LIN {X 0,Y 607.23,Z 1025.741,A -85,B 0,C 180,E1 27746.767,E2 27746.767} C_VEL
LIN {X 0,Y 605.649,Z 1047.101,A -85,B 0,C 180,E1 27745.787,E2 27745.787} C_VEL
LIN {X 0,Y 604.017,Z 1067.74,A -85,B 0,C 180,E1 27744.656,E2 27744.656} C_VEL
LIN {X 0,Y 602.404,Z 1085.974,A -85,B 0,C 180,E1 27743.476,E2 27743.476} C_VEL
LIN {X 0,Y 600.536,Z 1105.985,A -85,B 0,C 180,E1 27741.965,E2 27741.965} C_VEL
LIN {X 0,Y 598.945,Z 1123.019,A -85,B 0,C 180,E1 27740.472,E2 27740.472} C_VEL
LIN {X 0,Y 597.317,Z 1139.909,A -85,B 0,C 180,E1 27738.748,E2 27738.748} C_VEL
LIN {X 0,Y 595.864,Z 1155.688,A -85,B 0,C 180,E1 27736.876,E2 27736.876} C_VEL
LIN {X 0,Y 594.758,Z 1168.565,A -85,B 0,C 180,E1 27735.105,E2 27735.105} C_VEL
LIN {X 0,Y 593.832,Z 1180.293,A -85,B 0,C 180,E1 27733.238,E2 27733.238} C_VEL
LIN {X 0,Y 593.073,Z 1191.366,A -85,B 0,C 180,E1 27731.18,E2 27731.18} C_VEL
LIN {X 0,Y 592.512,Z 1201.281,A -85,B 0,C 180,E1 27728.932,E2 27728.932} C_VEL
LIN {X 0,Y 592.226,Z 1208.03,A -85,B 0,C 180,E1 27727.08,E2 27727.08} C_VEL
LIN {X 0,Y 592.061,Z 1213.419,A -85,B 0,C 180,E1 27725.33,E2 27725.33} C_VEL
LIN {X 0,Y 591.966,Z 1217.736,A -85,B 0,C 180,E1 27723.583,E2 27723.583} C_VEL
LIN {X 0,Y 591.922,Z 1221.023,A -85,B 0,C 180,E1 27721.839,E2 27721.839} C_VEL
LIN {X 0,Y 591.917,Z 1223.391,A -85,B 0,C 180,E1 27720,E2 27720} C_VEL
LIN {X 0,Y 591.915,Z 1224.654,A -85,B 0,C 180,E1 27718.161,E2 27718.161} C_VEL
LIN {X 0,Y 591.912,Z 1224.844,A -85,B 0,C 180,E1 27716.417,E2 27716.417} C_VEL
LIN {X 0,Y 591.911,Z 1224.051,A -85,B 0,C 180,E1 27714.669,E2 27714.669} C_VEL
LIN {X 0,Y 591.924,Z 1222.118,A -85,B 0,C 180,E1 27712.819,E2 27712.819} C_VEL
LIN {X 0,Y 591.947,Z 1219.241,A -85,B 0,C 180,E1 27711.06,E2 27711.06} C_VEL
LIN {X 0,Y 592.007,Z 1215.307,A -85,B 0,C 180,E1 27709.293,E2 27709.293} C_VEL
LIN {X 0,Y 592.15,Z 1210.275,A -85,B 0,C 180,E1 27707.518,E2 27707.518} C_VEL
LIN {X 0,Y 592.391,Z 1203.803,A -85,B 0,C 180,E1 27705.634,E2 27705.634} C_VEL
LIN {X 0,Y 592.739,Z 1196.926,A -85,B 0,C 180,E1 27703.939,E2 27703.939} C_VEL
LIN {X 0,Y 593.244,Z 1188.823,A -85,B 0,C 180,E1 27702.231,E2 27702.231} C_VEL
LIN {X 0,Y 594.061,Z 1177.572,A -85,B 0,C 180,E1 27700.201,E2 27700.201} C_VEL
LIN {X 0,Y 595.167,Z 1163.645,A -85,B 0,C 180,E1 27698.101,E2 27698.101} C_VEL
LIN {X 0,Y 596.308,Z 1150.164,A -85,B 0,C 180,E1 27696.374,E2 27696.374} C_VEL
LIN {X 0,Y 597.658,Z 1135.085,A -85,B 0,C 180,E1 27694.694,E2 27694.694} C_VEL
LIN {X 0,Y 599.006,Z 1119.589,A -85,B 0,C 180,E1 27693.211,E2 27693.211} C_VEL
LIN {X 0,Y 600.574,Z 1100.912,A -85,B 0,C 180,E1 27691.673,E2 27691.673} C_VEL
LIN {X 0,Y 602.005,Z 1082.997,A -85,B 0,C 180,E1 27690.411,E2 27690.411} C_VEL
LIN {X 0,Y 603.301,Z 1064.426,A -85,B 0,C 180,E1 27689.305,E2 27689.305} C_VEL
LIN {X 0,Y 604.533,Z 1044.81,A -85,B 0,C 180,E1 27688.307,E2 27688.307} C_VEL
LIN {X 0,Y 605.56,Z 1024.487,A -85,B 0,C 180,E1 27687.47,E2 27687.47} C_VEL
LIN {X 0,Y 606.425,Z 1002.632,A -85,B 0,C 180,E1 27686.742,E2 27686.742} C_VEL
LIN {X 0,Y 606.978,Z 981.871,A -85,B 0,C 180,E1 27686.218,E2 27686.218} C_VEL
LIN {X 0,Y 607.33,Z 958.537,A -85,B 0,C 180,E1 27685.807,E2 27685.807} C_VEL
LIN {X 0,Y 608.791,Z 782.484,A -85,B 0,C 180,E1 27683.738,E2 27683.738} C_VEL
LIN {X 0,Y 610.577,Z 662.5,A -85,B 0,C 180,E1 27682.165,E2 27682.165} C_VEL
LIN {X 0,Y 612.709,Z 661.282,A -85,B 0,C 180,E1 27681.912,E2 27681.912} C_VEL
LIN {X 0,Y 612.917,Z 662.99,A -85,B 0,C 180,E1 27681.212,E2 27681.212} C_VEL
LIN {X 0,Y 607.298,Z 672.97,A -85,B 0,C 180,E1 27679.896,E2 27679.896} C_VEL
LIN {X 0,Y 602.86,Z 684.875,A -85,B 0,C 180,E1 27678.563,E2 27678.563} C_VEL
LIN {X 0,Y 599.476,Z 698.903,A -85,B 0,C 180,E1 27677.215,E2 27677.215} C_VEL
LIN {X 0,Y 596.85,Z 716.647,A -85,B 0,C 180,E1 27675.741,E2 27675.741} C_VEL
LIN {X 0,Y 594.876,Z 740.159,A -85,B 0,C 180,E1 27674.033,E2 27674.033} C_VEL
LIN {X 0,Y 593.778,Z 772.685,A -85,B 0,C 180,E1 27671.9,E2 27671.9} C_VEL
LIN {X 0,Y 594.956,Z 795.605,A -85,B 0,C 180,E1 27670.446,E2 27670.446} C_VEL
LIN {X 0,Y 598.075,Z 815.31,A -85,B 0,C 180,E1 27669.196,E2 27669.196} C_VEL
LIN {X 0,Y 602.685,Z 831.753,A -85,B 0,C 180,E1 27668.15,E2 27668.15} C_VEL
LIN {X 0,Y 609.428,Z 848.007,A -85,B 0,C 180,E1 27667.119,E2 27667.119} C_VEL
LIN {X 0,Y 617.68,Z 862.679,A -85,B 0,C 180,E1 27666.199,E2 27666.199} C_VEL
LIN {X 0,Y 627.717,Z 876.404,A -85,B 0,C 180,E1 27665.356,E2 27665.356} C_VEL
LIN {X 0,Y 639.108,Z 888.723,A -85,B 0,C 180,E1 27664.62,E2 27664.62} C_VEL
LIN {X 0,Y 649.465,Z 898.016,A -85,B 0,C 180,E1 27664.084,E2 27664.084} C_VEL
LIN {X 0,Y 636.732,Z 910.076,A -85,B 0,C 180,E1 27663.45,E2 27663.45} C_VEL
LIN {X 0,Y 627.056,Z 921.639,A -85,B 0,C 180,E1 27662.823,E2 27662.823} C_VEL
LIN {X 0,Y 614.835,Z 940.901,A -85,B 0,C 180,E1 27661.751,E2 27661.751} C_VEL
LIN {X 0,Y 609.128,Z 960.233,A -85,B 0,C 180,E1 27661.71,E2 27661.71} C_VEL
LIN {X 0,Y 607.225,Z 972.37,A -85,B 0,C 180,E1 27661.624,E2 27661.624} C_VEL
LIN {X 0,Y 606.465,Z 1000.43,A -85,B 0,C 180,E1 27661.2,E2 27661.2} C_VEL
LIN {X 0,Y 605.336,Z 1030.279,A -85,B 0,C 180,E1 27660.57,E2 27660.57} C_VEL
LIN {X 0,Y 604.263,Z 1057.387,A -85,B 0,C 180,E1 27659.82,E2 27659.82} C_VEL
LIN {X 0,Y 603.092,Z 1083.908,A -85,B 0,C 180,E1 27658.908,E2 27658.908} C_VEL
LIN {X 0,Y 601.89,Z 1109.704,A -85,B 0,C 180,E1 27657.829,E2 27657.829} C_VEL
LIN {X 0,Y 600.679,Z 1133.526,A -85,B 0,C 180,E1 27656.633,E2 27656.633} C_VEL
LIN {X 0,Y 599.46,Z 1155.536,A -85,B 0,C 180,E1 27655.331,E2 27655.331} C_VEL
LIN {X 0,Y 598.296,Z 1175.247,A -85,B 0,C 180,E1 27653.962,E2 27653.962} C_VEL
LIN {X 0,Y 597.307,Z 1190.761,A -85,B 0,C 180,E1 27652.724,E2 27652.724} C_VEL
LIN {X 0,Y 596.459,Z 1203.994,A -85,B 0,C 180,E1 27651.54,E2 27651.54} C_VEL
LIN {X 0,Y 595.623,Z 1216.939,A -85,B 0,C 180,E1 27650.233,E2 27650.233} C_VEL
LIN {X 0,Y 594.889,Z 1228.403,A -85,B 0,C 180,E1 27648.93,E2 27648.93} C_VEL
LIN {X 0,Y 594.202,Z 1239.278,A -85,B 0,C 180,E1 27647.531,E2 27647.531} C_VEL
LIN {X 0,Y 593.59,Z 1249.466,A -85,B 0,C 180,E1 27646.038,E2 27646.038} C_VEL
LIN {X 0,Y 593.111,Z 1258.344,A -85,B 0,C 180,E1 27644.549,E2 27644.549} C_VEL
LIN {X 0,Y 592.688,Z 1266.505,A -85,B 0,C 180,E1 27642.967,E2 27642.967} C_VEL
LIN {X 0,Y 592.393,Z 1273.427,A -85,B 0,C 180,E1 27641.391,E2 27641.391} C_VEL
LIN {X 0,Y 592.174,Z 1279.691,A -85,B 0,C 180,E1 27639.624,E2 27639.624} C_VEL
LIN {X 0,Y 592.016,Z 1284.794,A -85,B 0,C 180,E1 27637.864,E2 27637.864} C_VEL
LIN {X 0,Y 591.951,Z 1288.822,A -85,B 0,C 180,E1 27636.11,E2 27636.11} C_VEL
LIN {X 0,Y 591.912,Z 1291.811,A -85,B 0,C 180,E1 27634.361,E2 27634.361} C_VEL
LIN {X 0,Y 591.897,Z 1293.788,A -85,B 0,C 180,E1 27632.616,E2 27632.616} C_VEL
LIN {X 0,Y 591.9,Z 1294.798,A -85,B 0,C 180,E1 27630.776,E2 27630.776} C_VEL
LIN {X 0,Y 591.908,Z 1294.739,A -85,B 0,C 180,E1 27629.033,E2 27629.033} C_VEL
LIN {X 0,Y 591.901,Z 1293.621,A -85,B 0,C 180,E1 27627.193,E2 27627.193} C_VEL
LIN {X 0,Y 591.911,Z 1291.258,A -85,B 0,C 180,E1 27625.253,E2 27625.253} C_VEL
LIN {X 0,Y 591.98,Z 1286.809,A -85,B 0,C 180,E1 27622.919,E2 27622.919} C_VEL
LIN {X 0,Y 592.119,Z 1280.934,A -85,B 0,C 180,E1 27620.77,E2 27620.77} C_VEL
LIN {X 0,Y 592.336,Z 1274.94,A -85,B 0,C 180,E1 27619.005,E2 27619.005} C_VEL
LIN {X 0,Y 592.629,Z 1267.976,A -85,B 0,C 180,E1 27617.331,E2 27617.331} C_VEL
LIN {X 0,Y 593.049,Z 1259.769,A -85,B 0,C 180,E1 27615.652,E2 27615.652} C_VEL
LIN {X 0,Y 593.593,Z 1250.249,A -85,B 0,C 180,E1 27613.965,E2 27613.965} C_VEL
LIN {X 0,Y 594.356,Z 1238.884,A -85,B 0,C 180,E1 27612.212,E2 27612.212} C_VEL
LIN {X 0,Y 595.465,Z 1223.553,A -85,B 0,C 180,E1 27610.174,E2 27610.174} C_VEL
LIN {X 0,Y 596.638,Z 1208.398,A -85,B 0,C 180,E1 27608.453,E2 27608.453} C_VEL
LIN {X 0,Y 597.954,Z 1192.476,A -85,B 0,C 180,E1 27606.863,E2 27606.863} C_VEL
LIN {X 0,Y 599.507,Z 1174.108,A -85,B 0,C 180,E1 27605.254,E2 27605.254} C_VEL
LIN {X 0,Y 601.35,Z 1152.649,A -85,B 0,C 180,E1 27603.646,E2 27603.646} C_VEL
LIN {X 0,Y 603.159,Z 1131.512,A -85,B 0,C 180,E1 27602.282,E2 27602.282} C_VEL
LIN {X 0,Y 604.976,Z 1109.76,A -85,B 0,C 180,E1 27601.092,E2 27601.092} C_VEL
LIN {X 0,Y 606.798,Z 1087.393,A -85,B 0,C 180,E1 27600.049,E2 27600.049} C_VEL
LIN {X 0,Y 608.552,Z 1064.048,A -85,B 0,C 180,E1 27599.162,E2 27599.162} C_VEL
LIN {X 0,Y 610.274,Z 1039.967,A -85,B 0,C 180,E1 27598.426,E2 27598.426} C_VEL
LIN {X 0,Y 611.681,Z 1016.352,A -85,B 0,C 180,E1 27597.883,E2 27597.883} C_VEL
LIN {X 0,Y 612.739,Z 990.04,A -85,B 0,C 180,E1 27597.453,E2 27597.453} C_VEL
LIN {X 0,Y 613.619,Z 969.904,A -85,B 0,C 180,E1 27597.188,E2 27597.188} C_VEL
LIN {X 0,Y 614.818,Z 961.81,A -85,B 0,C 180,E1 27597.101,E2 27597.101} C_VEL
LIN {X 0,Y 620.981,Z 950.092,A -85,B 0,C 180,E1 27596.478,E2 27596.478} C_VEL
LIN {X 0,Y 631.79,Z 932.766,A -85,B 0,C 180,E1 27595.655,E2 27595.655} C_VEL
LIN {X 0,Y 641.465,Z 920.212,A -85,B 0,C 180,E1 27595.162,E2 27595.162} C_VEL
LIN {X 0,Y 652.853,Z 907.547,A -85,B 0,C 180,E1 27594.757,E2 27594.757} C_VEL
LIN {X 0,Y 641.985,Z 899.958,A -85,B 0,C 180,E1 27593.633,E2 27593.633} C_VEL
LIN {X 0,Y 632.323,Z 890.651,A -85,B 0,C 180,E1 27592.385,E2 27592.385} C_VEL
LIN {X 0,Y 624.741,Z 880.508,A -85,B 0,C 180,E1 27591.144,E2 27591.144} C_VEL
LIN {X 0,Y 618.586,Z 868.552,A -85,B 0,C 180,E1 27589.797,E2 27589.797} C_VEL
LIN {X 0,Y 614.2,Z 855.239,A -85,B 0,C 180,E1 27588.415,E2 27588.415} C_VEL
LIN {X 0,Y 611.769,Z 840.893,A -85,B 0,C 180,E1 27587.037,E2 27587.037} C_VEL
LIN {X 0,Y 611.126,Z 822.711,A -85,B 0,C 180,E1 27585.423,E2 27585.423} C_VEL
LIN {X 0,Y 614.294,Z 776.645,A -85,B 0,C 180,E1 27581.571,E2 27581.571} C_VEL
LIN {X 0,Y 617.028,Z 740.676,A -85,B 0,C 180,E1 27578.495,E2 27578.495} C_VEL
LIN {X 0,Y 619.611,Z 706.77,A -85,B 0,C 180,E1 27575.517,E2 27575.517} C_VEL
LIN {X 0,Y 621.707,Z 679.327,A -85,B 0,C 180,E1 27573.039,E2 27573.039} C_VEL
LIN {X 0,Y 613.464,Z 659.709,A -85,B 0,C 180,E1 27570.241,E2 27570.241} C_VEL
LIN {X 0,Y 605.961,Z 642.448,A -85,B 0,C 180,E1 27567.617,E2 27567.617} C_VEL
LIN {X 0,Y 598.637,Z 626.33,A -85,B 0,C 180,E1 27564.998,E2 27564.998} C_VEL
LIN {X 0,Y 594.504,Z 617.583,A -85,B 0,C 180,E1 27563.491,E2 27563.491} C_VEL
LIN {X 0,Y 593.187,Z 614.089,A -85,B 0,C 180,E1 27562.916,E2 27562.916} C_VEL
LIN {X 0,Y 593.198,Z 614.092,A -85,B 0,C 180,E1 27559.702,E2 27559.702} C_VEL
LIN {X 0,Y 593.192,Z 614.089,A -85,B 0,C 180,E1 27556.449,E2 27556.449} C_VEL
LIN {X 0,Y 593.2,Z 614.086,A -85,B 0,C 180,E1 27553.252,E2 27553.252} C_VEL
LIN {X 0,Y 593.195,Z 614.089,A -85,B 0,C 180,E1 27549.998,E2 27549.998} C_VEL
LIN {X 0,Y 593.202,Z 614.086,A -85,B 0,C 180,E1 27546.776,E2 27546.776} C_VEL
LIN {X 0,Y 593.188,Z 614.087,A -85,B 0,C 180,E1 27543.479,E2 27543.479} C_VEL
LIN {X 0,Y 593.191,Z 614.091,A -85,B 0,C 180,E1 27540.29,E2 27540.29} C_VEL
LIN {X 0,Y 593.185,Z 614.093,A -85,B 0,C 180,E1 27537.101,E2 27537.101} C_VEL
LIN {X 0,Y 593.19,Z 614.091,A -85,B 0,C 180,E1 27533.904,E2 27533.904} C_VEL
LIN {X 0,Y 593.18,Z 614.09,A -85,B 0,C 180,E1 27530.687,E2 27530.687} C_VEL
LIN {X 0,Y 593.192,Z 614.087,A -85,B 0,C 180,E1 27527.441,E2 27527.441} C_VEL
LIN {X 0,Y 593.184,Z 614.089,A -85,B 0,C 180,E1 27524.251,E2 27524.251} C_VEL
LIN {X 0,Y 593.199,Z 614.088,A -85,B 0,C 180,E1 27521.01,E2 27521.01} C_VEL
LIN {X 0,Y 593.201,Z 614.087,A -85,B 0,C 180,E1 27517.608,E2 27517.608} C_VEL
LIN {X 0,Y 593.191,Z 614.089,A -85,B 0,C 180,E1 27514.329,E2 27514.329} C_VEL
LIN {X 0,Y 593.183,Z 614.09,A -85,B 0,C 180,E1 27511.067,E2 27511.067} C_VEL
LIN {X 0,Y 593.185,Z 614.088,A -85,B 0,C 180,E1 27507.929,E2 27507.929} C_VEL
LIN {X 0,Y 593.182,Z 614.083,A -85,B 0,C 180,E1 27504.796,E2 27504.796} C_VEL
LIN {X 0,Y 593.181,Z 614.084,A -85,B 0,C 180,E1 27501.609,E2 27501.609} C_VEL
LIN {X 0,Y 593.182,Z 614.086,A -85,B 0,C 180,E1 27498.451,E2 27498.451} C_VEL
LIN {X 0,Y 593.183,Z 614.084,A -85,B 0,C 180,E1 27495.203,E2 27495.203} C_VEL
LIN {X 0,Y 593.181,Z 614.076,A -85,B 0,C 180,E1 27491.98,E2 27491.98} C_VEL
LIN {X 0,Y 593.184,Z 614.094,A -85,B 0,C 180,E1 27488.831,E2 27488.831} C_VEL
LIN {X 0,Y 593.19,Z 614.096,A -85,B 0,C 180,E1 27485.557,E2 27485.557} C_VEL
LIN {X 0,Y 593.192,Z 614.166,A -85,B 0,C 180,E1 27483.94,E2 27483.94} C_VEL
LIN {X 0,Y 601.823,Z 640.811,A -85,B 0,C 180,E1 27481.667,E2 27481.667} C_VEL
LIN {X 0,Y 603.521,Z 647.357,A -85,B 0,C 180,E1 27481.123,E2 27481.123} C_VEL
LIN {X 0,Y 602.85,Z 675.783,A -85,B 0,C 180,E1 27479.149,E2 27479.149} C_VEL
LIN {X 0,Y 601.769,Z 682.206,A -85,B 0,C 180,E1 27478.744,E2 27478.744} C_VEL
LIN {X 0,Y 595.436,Z 699.841,A -85,B 0,C 180,E1 27477.78,E2 27477.78} C_VEL
LIN {X 0,Y 594.571,Z 705.297,A -85,B 0,C 180,E1 27477.423,E2 27477.423} C_VEL
LIN {X 0,Y 593.027,Z 749.74,A -85,B 0,C 180,E1 27474.26,E2 27474.26} C_VEL
LIN {X 0,Y 591.603,Z 795.59,A -85,B 0,C 180,E1 27471.047,E2 27471.047} C_VEL
LIN {X 0,Y 590.598,Z 840.977,A -85,B 0,C 180,E1 27468.002,E2 27468.002} C_VEL
LIN {X 0,Y 591.441,Z 849.835,A -85,B 0,C 180,E1 27467.861,E2 27467.861} C_VEL
LIN {X 0,Y 589.997,Z 1011.072,A -85,B 0,C 180,E1 27465.855,E2 27465.855} C_VEL
LIN {X 0,Y 589.774,Z 1028.498,A -85,B 0,C 180,E1 27465.459,E2 27465.459} C_VEL
LIN {X 0,Y 589.357,Z 1045.18,A -85,B 0,C 180,E1 27464.892,E2 27464.892} C_VEL
LIN {X 0,Y 588.801,Z 1061.441,A -85,B 0,C 180,E1 27464.148,E2 27464.148} C_VEL
LIN {X 0,Y 588.166,Z 1076.49,A -85,B 0,C 180,E1 27463.266,E2 27463.266} C_VEL
LIN {X 0,Y 587.477,Z 1090.538,A -85,B 0,C 180,E1 27462.232,E2 27462.232} C_VEL
LIN {X 0,Y 586.768,Z 1103.789,A -85,B 0,C 180,E1 27461.024,E2 27461.024} C_VEL
LIN {X 0,Y 586.126,Z 1115.428,A -85,B 0,C 180,E1 27459.722,E2 27459.722} C_VEL
LIN {X 0,Y 585.586,Z 1125.434,A -85,B 0,C 180,E1 27458.344,E2 27458.344} C_VEL
LIN {X 0,Y 585.142,Z 1133.991,A -85,B 0,C 180,E1 27456.868,E2 27456.868} C_VEL
LIN {X 0,Y 584.803,Z 1141.524,A -85,B 0,C 180,E1 27455.198,E2 27455.198} C_VEL
LIN {X 0,Y 584.593,Z 1147.073,A -85,B 0,C 180,E1 27453.529,E2 27453.529} C_VEL
LIN {X 0,Y 584.464,Z 1150.768,A -85,B 0,C 180,E1 27451.861,E2 27451.861} C_VEL
LIN {X 0,Y 584.417,Z 1152.844,A -85,B 0,C 180,E1 27450.097,E2 27450.097} C_VEL
LIN {X 0,Y 584.398,Z 1153.14,A -85,B 0,C 180,E1 27448.332,E2 27448.332} C_VEL
LIN {X 0,Y 584.444,Z 1151.759,A -85,B 0,C 180,E1 27446.664,E2 27446.664} C_VEL
LIN {X 0,Y 584.541,Z 1148.673,A -85,B 0,C 180,E1 27444.994,E2 27444.994} C_VEL
LIN {X 0,Y 584.725,Z 1143.83,A -85,B 0,C 180,E1 27443.321,E2 27443.321} C_VEL
LIN {X 0,Y 585.02,Z 1137.091,A -85,B 0,C 180,E1 27441.645,E2 27441.645} C_VEL
LIN {X 0,Y 585.41,Z 1129.301,A -85,B 0,C 180,E1 27440.164,E2 27440.164} C_VEL
LIN {X 0,Y 585.938,Z 1119.419,A -85,B 0,C 180,E1 27438.681,E2 27438.681} C_VEL
LIN {X 0,Y 586.588,Z 1107.969,A -85,B 0,C 180,E1 27437.296,E2 27437.296} C_VEL
LIN {X 0,Y 587.259,Z 1095.915,A -85,B 0,C 180,E1 27436.108,E2 27436.108} C_VEL
LIN {X 0,Y 587.97,Z 1082.071,A -85,B 0,C 180,E1 27435.002,E2 27435.002} C_VEL
LIN {X 0,Y 588.658,Z 1066.841,A -85,B 0,C 180,E1 27434.027,E2 27434.027} C_VEL
LIN {X 0,Y 589.259,Z 1051.079,A -85,B 0,C 180,E1 27433.233,E2 27433.233} C_VEL
LIN {X 0,Y 589.73,Z 1034.418,A -85,B 0,C 180,E1 27432.602,E2 27432.602} C_VEL
LIN {X 0,Y 590.029,Z 1016.924,A -85,B 0,C 180,E1 27432.14,E2 27432.14} C_VEL
LIN {X 0,Y 590.161,Z 997.63,A -85,B 0,C 180,E1 27431.834,E2 27431.834} C_VEL
LIN {X 0,Y 591.377,Z 845.871,A -85,B 0,C 180,E1 27429.959,E2 27429.959} C_VEL
LIN {X 0,Y 590.71,Z 840.625,A -85,B 0,C 180,E1 27429.85,E2 27429.85} C_VEL
LIN {X 0,Y 591.797,Z 794.074,A -85,B 0,C 180,E1 27426.71,E2 27426.71} C_VEL
LIN {X 0,Y 593.303,Z 748.165,A -85,B 0,C 180,E1 27423.473,E2 27423.473} C_VEL
LIN {X 0,Y 594.871,Z 704.382,A -85,B 0,C 180,E1 27420.343,E2 27420.343} C_VEL
LIN {X 0,Y 596.219,Z 662.017,A -85,B 0,C 180,E1 27417.34,E2 27417.34} C_VEL
LIN {X 0,Y 596.383,Z 649.162,A -85,B 0,C 180,E1 27416.436,E2 27416.436} C_VEL
LIN {X 0,Y 588.994,Z 625.935,A -85,B 0,C 180,E1 27414.406,E2 27414.406} C_VEL
LIN {X 0,Y 585.252,Z 615.062,A -85,B 0,C 180,E1 27413.417,E2 27413.417} C_VEL
LIN {X 0,Y 585.244,Z 615.057,A -85,B 0,C 180,E1 27410.156,E2 27410.156} C_VEL
LIN {X 0,Y 585.252,Z 615.076,A -85,B 0,C 180,E1 27406.99,E2 27406.99} C_VEL
LIN {X 0,Y 585.247,Z 615.08,A -85,B 0,C 180,E1 27403.722,E2 27403.722} C_VEL
LIN {X 0,Y 585.243,Z 615.077,A -85,B 0,C 180,E1 27400.484,E2 27400.484} C_VEL
LIN {X 0,Y 585.257,Z 615.077,A -85,B 0,C 180,E1 27397.236,E2 27397.236} C_VEL
LIN {X 0,Y 585.28,Z 615.26,A -85,B 0,C 180,E1 27396.914,E2 27396.914} C_VEL
LIN {X 0,Y 586.619,Z 618.666,A -85,B 0,C 180,E1 27396.435,E2 27396.435} C_VEL
LIN {X 0,Y 589.325,Z 624.916,A -85,B 0,C 180,E1 27395.584,E2 27395.584} C_VEL
LIN {X 0,Y 604.455,Z 647.067,A -85,B 0,C 180,E1 27394.049,E2 27394.049} C_VEL
LIN {X 0,Y 611.334,Z 657.936,A -85,B 0,C 180,E1 27393.366,E2 27393.366} C_VEL
LIN {X 0,Y 604.902,Z 898.8,A -85,B 0,C 180,E1 27389.957,E2 27389.957} C_VEL
LIN {X 0,Y 603.542,Z 958.961,A -85,B 0,C 180,E1 27389.101,E2 27389.101} C_VEL
LIN {X 0,Y 602.63,Z 981.844,A -85,B 0,C 180,E1 27388.598,E2 27388.598} C_VEL
LIN {X 0,Y 601.437,Z 1005.236,A -85,B 0,C 180,E1 27387.904,E2 27387.904} C_VEL
LIN {X 0,Y 600.19,Z 1025.082,A -85,B 0,C 180,E1 27387.16,E2 27387.16} C_VEL
LIN {X 0,Y 598.533,Z 1046.708,A -85,B 0,C 180,E1 27386.17,E2 27386.17} C_VEL
LIN {X 0,Y 596.816,Z 1067.535,A -85,B 0,C 180,E1 27385.026,E2 27385.026} C_VEL
LIN {X 0,Y 595.052,Z 1086.552,A -85,B 0,C 180,E1 27383.784,E2 27383.784} C_VEL
LIN {X 0,Y 593.127,Z 1106.143,A -85,B 0,C 180,E1 27382.291,E2 27382.291} C_VEL
LIN {X 0,Y 591.419,Z 1123.556,A -85,B 0,C 180,E1 27380.749,E2 27380.749} C_VEL
LIN {X 0,Y 589.776,Z 1139.554,A -85,B 0,C 180,E1 27379.099,E2 27379.099} C_VEL
LIN {X 0,Y 588.319,Z 1154.745,A -85,B 0,C 180,E1 27377.303,E2 27377.303} C_VEL
LIN {X 0,Y 587.039,Z 1168.49,A -85,B 0,C 180,E1 27375.407,E2 27375.407} C_VEL
LIN {X 0,Y 585.957,Z 1181.443,A -85,B 0,C 180,E1 27373.319,E2 27373.319} C_VEL
LIN {X 0,Y 585.093,Z 1193.321,A -85,B 0,C 180,E1 27371.035,E2 27371.035} C_VEL
LIN {X 0,Y 584.567,Z 1202.221,A -85,B 0,C 180,E1 27368.955,E2 27368.955} C_VEL
LIN {X 0,Y 584.246,Z 1209.26,A -85,B 0,C 180,E1 27366.96,E2 27366.96} C_VEL
LIN {X 0,Y 584.065,Z 1214.56,A -85,B 0,C 180,E1 27365.107,E2 27365.107} C_VEL
LIN {X 0,Y 583.966,Z 1218.563,A -85,B 0,C 180,E1 27363.337,E2 27363.337} C_VEL
LIN {X 0,Y 583.919,Z 1221.56,A -85,B 0,C 180,E1 27361.57,E2 27361.57} C_VEL
LIN {X 0,Y 583.91,Z 1223.69,A -85,B 0,C 180,E1 27359.706,E2 27359.706} C_VEL
LIN {X 0,Y 583.908,Z 1224.728,A -85,B 0,C 180,E1 27357.939,E2 27357.939} C_VEL
LIN {X 0,Y 583.914,Z 1224.783,A -85,B 0,C 180,E1 27356.171,E2 27356.171} C_VEL
LIN {X 0,Y 583.913,Z 1223.931,A -85,B 0,C 180,E1 27354.497,E2 27354.497} C_VEL
LIN {X 0,Y 583.923,Z 1221.95,A -85,B 0,C 180,E1 27352.621,E2 27352.621} C_VEL
LIN {X 0,Y 583.96,Z 1219.088,A -85,B 0,C 180,E1 27350.837,E2 27350.837} C_VEL
LIN {X 0,Y 584.038,Z 1215.197,A -85,B 0,C 180,E1 27349.045,E2 27349.045} C_VEL
LIN {X 0,Y 584.207,Z 1210.229,A -85,B 0,C 180,E1 27347.245,E2 27347.245} C_VEL
LIN {X 0,Y 584.521,Z 1203.359,A -85,B 0,C 180,E1 27345.233,E2 27345.233} C_VEL
LIN {X 0,Y 585.075,Z 1194.047,A -85,B 0,C 180,E1 27343.008,E2 27343.008} C_VEL
LIN {X 0,Y 585.847,Z 1183.062,A -85,B 0,C 180,E1 27340.871,E2 27340.871} C_VEL
LIN {X 0,Y 586.856,Z 1170.602,A -85,B 0,C 180,E1 27338.826,E2 27338.826} C_VEL
LIN {X 0,Y 587.938,Z 1158.168,A -85,B 0,C 180,E1 27337.079,E2 27337.079} C_VEL
LIN {X 0,Y 589.304,Z 1143.221,A -85,B 0,C 180,E1 27335.276,E2 27335.276} C_VEL
LIN {X 0,Y 590.716,Z 1127.908,A -85,B 0,C 180,E1 27333.674,E2 27333.674} C_VEL
LIN {X 0,Y 592.227,Z 1111.048,A -85,B 0,C 180,E1 27332.171,E2 27332.171} C_VEL
LIN {X 0,Y 593.773,Z 1092.835,A -85,B 0,C 180,E1 27330.768,E2 27330.768} C_VEL
LIN {X 0,Y 595.133,Z 1075.358,A -85,B 0,C 180,E1 27329.621,E2 27329.621} C_VEL
LIN {X 0,Y 596.579,Z 1054.641,A -85,B 0,C 180,E1 27328.471,E2 27328.471} C_VEL
LIN {X 0,Y 597.675,Z 1035.647,A -85,B 0,C 180,E1 27327.592,E2 27327.592} C_VEL
LIN {X 0,Y 598.649,Z 1014.559,A -85,B 0,C 180,E1 27326.804,E2 27326.804} C_VEL
LIN {X 0,Y 599.393,Z 992.898,A -85,B 0,C 180,E1 27326.165,E2 27326.165} C_VEL
LIN {X 0,Y 599.828,Z 971.457,A -85,B 0,C 180,E1 27325.713,E2 27325.713} C_VEL
LIN {X 0,Y 600.05,Z 943.563,A -85,B 0,C 180,E1 27325.33,E2 27325.33} C_VEL
LIN {X 0,Y 601.341,Z 803.115,A -85,B 0,C 180,E1 27323.666,E2 27323.666} C_VEL
LIN {X 0,Y 603.148,Z 687.762,A -85,B 0,C 180,E1 27322.133,E2 27322.133} C_VEL
LIN {X 0,Y 603.687,Z 668.604,A -85,B 0,C 180,E1 27321.844,E2 27321.844} C_VEL
LIN {X 0,Y 606.072,Z 667.295,A -85,B 0,C 180,E1 27321.597,E2 27321.597} C_VEL
LIN {X 0,Y 606.566,Z 667.049,A -85,B 0,C 180,E1 27321.538,E2 27321.538} C_VEL
LIN {X 0,Y 600.941,Z 676.357,A -85,B 0,C 180,E1 27320.239,E2 27320.239} C_VEL
LIN {X 0,Y 596.232,Z 687.752,A -85,B 0,C 180,E1 27318.899,E2 27318.899} C_VEL
LIN {X 0,Y 592.53,Z 701.469,A -85,B 0,C 180,E1 27317.514,E2 27317.514} C_VEL
LIN {X 0,Y 589.682,Z 718.28,A -85,B 0,C 180,E1 27316.046,E2 27316.046} C_VEL
LIN {X 0,Y 587.46,Z 740.787,A -85,B 0,C 180,E1 27314.33,E2 27314.33} C_VEL
LIN {X 0,Y 586.076,Z 771.491,A -85,B 0,C 180,E1 27312.231,E2 27312.231} C_VEL
LIN {X 0,Y 586.946,Z 794.766,A -85,B 0,C 180,E1 27310.705,E2 27310.705} C_VEL
LIN {X 0,Y 589.869,Z 815.078,A -85,B 0,C 180,E1 27309.378,E2 27309.378} C_VEL
LIN {X 0,Y 594.509,Z 832.549,A -85,B 0,C 180,E1 27308.239,E2 27308.239} C_VEL
LIN {X 0,Y 601.076,Z 848.949,A -85,B 0,C 180,E1 27307.172,E2 27307.172} C_VEL
LIN {X 0,Y 608.923,Z 863.473,A -85,B 0,C 180,E1 27306.239,E2 27306.239} C_VEL
LIN {X 0,Y 618.214,Z 876.831,A -85,B 0,C 180,E1 27305.396,E2 27305.396} C_VEL
LIN {X 0,Y 629.342,Z 889.591,A -85,B 0,C 180,E1 27304.614,E2 27304.614} C_VEL
LIN {X 0,Y 638.146,Z 898.311,A -85,B 0,C 180,E1 27304.097,E2 27304.097} C_VEL
LIN {X 0,Y 626.508,Z 910.311,A -85,B 0,C 180,E1 27303.465,E2 27303.465} C_VEL
LIN {X 0,Y 617.586,Z 921.928,A -85,B 0,C 180,E1 27302.83,E2 27302.83} C_VEL
LIN {X 0,Y 608.578,Z 936.477,A -85,B 0,C 180,E1 27302.039,E2 27302.039} C_VEL
LIN {X 0,Y 602.917,Z 954.76,A -85,B 0,C 180,E1 27302.018,E2 27302.018} C_VEL
LIN {X 0,Y 600.287,Z 967.685,A -85,B 0,C 180,E1 27301.95,E2 27301.95} C_VEL
LIN {X 0,Y 599.475,Z 980.408,A -85,B 0,C 180,E1 27301.793,E2 27301.793} C_VEL
LIN {X 0,Y 598.514,Z 1010.495,A -85,B 0,C 180,E1 27301.244,E2 27301.244} C_VEL
LIN {X 0,Y 597.304,Z 1039.086,A -85,B 0,C 180,E1 27300.55,E2 27300.55} C_VEL
LIN {X 0,Y 596.078,Z 1066.15,A -85,B 0,C 180,E1 27299.716,E2 27299.716} C_VEL
LIN {X 0,Y 594.868,Z 1092.154,A -85,B 0,C 180,E1 27298.734,E2 27298.734} C_VEL
LIN {X 0,Y 593.642,Z 1117.256,A -85,B 0,C 180,E1 27297.594,E2 27297.594} C_VEL
LIN {X 0,Y 592.335,Z 1140.975,A -85,B 0,C 180,E1 27296.316,E2 27296.316} C_VEL
LIN {X 0,Y 591.061,Z 1163.061,A -85,B 0,C 180,E1 27294.913,E2 27294.913} C_VEL
LIN {X 0,Y 589.773,Z 1183.661,A -85,B 0,C 180,E1 27293.374,E2 27293.374} C_VEL
LIN {X 0,Y 588.65,Z 1201.31,A -85,B 0,C 180,E1 27291.84,E2 27291.84} C_VEL
LIN {X 0,Y 587.702,Z 1215.852,A -85,B 0,C 180,E1 27290.372,E2 27290.372} C_VEL
LIN {X 0,Y 586.915,Z 1227.948,A -85,B 0,C 180,E1 27288.991,E2 27288.991} C_VEL
LIN {X 0,Y 586.218,Z 1238.906,A -85,B 0,C 180,E1 27287.573,E2 27287.573} C_VEL
LIN {X 0,Y 585.598,Z 1249.162,A -85,B 0,C 180,E1 27286.059,E2 27286.059} C_VEL
LIN {X 0,Y 585.115,Z 1258.094,A -85,B 0,C 180,E1 27284.55,E2 27284.55} C_VEL
LIN {X 0,Y 584.689,Z 1266.292,A -85,B 0,C 180,E1 27282.947,E2 27282.947} C_VEL
LIN {X 0,Y 584.391,Z 1273.283,A -85,B 0,C 180,E1 27281.349,E2 27281.349} C_VEL
LIN {X 0,Y 584.176,Z 1279.576,A -85,B 0,C 180,E1 27279.632,E2 27279.632} C_VEL
LIN {X 0,Y 584.021,Z 1284.565,A -85,B 0,C 180,E1 27277.973,E2 27277.973} C_VEL
LIN {X 0,Y 583.958,Z 1288.775,A -85,B 0,C 180,E1 27276.194,E2 27276.194} C_VEL
LIN {X 0,Y 583.91,Z 1291.671,A -85,B 0,C 180,E1 27274.519,E2 27274.519} C_VEL
LIN {X 0,Y 583.899,Z 1293.703,A -85,B 0,C 180,E1 27272.75,E2 27272.75} C_VEL
LIN {X 0,Y 583.908,Z 1294.742,A -85,B 0,C 180,E1 27270.983,E2 27270.983} C_VEL
LIN {X 0,Y 583.901,Z 1294.791,A -85,B 0,C 180,E1 27269.216,E2 27269.216} C_VEL
LIN {X 0,Y 583.897,Z 1293.863,A -85,B 0,C 180,E1 27267.45,E2 27267.45} C_VEL
LIN {X 0,Y 583.913,Z 1291.943,A -85,B 0,C 180,E1 27265.68,E2 27265.68} C_VEL
LIN {X 0,Y 583.942,Z 1289.175,A -85,B 0,C 180,E1 27264.006,E2 27264.006} C_VEL
LIN {X 0,Y 584.012,Z 1285.129,A -85,B 0,C 180,E1 27262.228,E2 27262.228} C_VEL
LIN {X 0,Y 584.166,Z 1279.952,A -85,B 0,C 180,E1 27260.444,E2 27260.444} C_VEL
LIN {X 0,Y 584.367,Z 1273.969,A -85,B 0,C 180,E1 27258.753,E2 27258.753} C_VEL
LIN {X 0,Y 584.684,Z 1266.853,A -85,B 0,C 180,E1 27257.056,E2 27257.056} C_VEL
LIN {X 0,Y 585.171,Z 1257.995,A -85,B 0,C 180,E1 27255.252,E2 27255.252} C_VEL
LIN {X 0,Y 585.909,Z 1246.304,A -85,B 0,C 180,E1 27253.213,E2 27253.213} C_VEL
LIN {X 0,Y 586.919,Z 1231.939,A -85,B 0,C 180,E1 27251.116,E2 27251.116} C_VEL
LIN {X 0,Y 587.995,Z 1218.309,A -85,B 0,C 180,E1 27249.392,E2 27249.392} C_VEL
LIN {X 0,Y 589.338,Z 1202.321,A -85,B 0,C 180,E1 27247.619,E2 27247.619} C_VEL
LIN {X 0,Y 591.071,Z 1182.47,A -85,B 0,C 180,E1 27245.73,E2 27245.73} C_VEL
LIN {X 0,Y 592.813,Z 1163.203,A -85,B 0,C 180,E1 27244.152,E2 27244.152} C_VEL
LIN {X 0,Y 594.712,Z 1142.5,A -85,B 0,C 180,E1 27242.68,E2 27242.68} C_VEL
LIN {X 0,Y 596.574,Z 1121.597,A -85,B 0,C 180,E1 27241.414,E2 27241.414} C_VEL
LIN {X 0,Y 598.548,Z 1099.427,A -85,B 0,C 180,E1 27240.257,E2 27240.257} C_VEL
LIN {X 0,Y 600.373,Z 1077.489,A -85,B 0,C 180,E1 27239.308,E2 27239.308} C_VEL
LIN {X 0,Y 602.248,Z 1054.203,A -85,B 0,C 180,E1 27238.47,E2 27238.47} C_VEL
LIN {X 0,Y 603.92,Z 1030.402,A -85,B 0,C 180,E1 27237.806,E2 27237.806} C_VEL
LIN {X 0,Y 605.446,Z 1005.337,A -85,B 0,C 180,E1 27237.284,E2 27237.284} C_VEL
LIN {X 0,Y 606.827,Z 971.213,A -85,B 0,C 180,E1 27236.786,E2 27236.786} C_VEL
LIN {X 0,Y 608.167,Z 960.66,A -85,B 0,C 180,E1 27236.695,E2 27236.695} C_VEL
LIN {X 0,Y 614.389,Z 948.944,A -85,B 0,C 180,E1 27236.07,E2 27236.07} C_VEL
LIN {X 0,Y 625.665,Z 930.976,A -85,B 0,C 180,E1 27235.215,E2 27235.215} C_VEL
LIN {X 0,Y 635.328,Z 918.412,A -85,B 0,C 180,E1 27234.721,E2 27234.721} C_VEL
LIN {X 0,Y 642.556,Z 910.034,A -85,B 0,C 180,E1 27234.438,E2 27234.438} C_VEL
LIN {X 0,Y 632.379,Z 902.013,A -85,B 0,C 180,E1 27233.288,E2 27233.288} C_VEL
LIN {X 0,Y 623.114,Z 892.094,A -85,B 0,C 180,E1 27231.989,E2 27231.989} C_VEL
LIN {X 0,Y 616.103,Z 881.582,A -85,B 0,C 180,E1 27230.727,E2 27230.727} C_VEL
LIN {X 0,Y 610.327,Z 869.05,A -85,B 0,C 180,E1 27229.335,E2 27229.335} C_VEL
LIN {X 0,Y 606.377,Z 855.129,A -85,B 0,C 180,E1 27227.905,E2 27227.905} C_VEL
LIN {X 0,Y 604.358,Z 839.729,A -85,B 0,C 180,E1 27226.441,E2 27226.441} C_VEL
LIN {X 0,Y 604.25,Z 820.8,A -85,B 0,C 180,E1 27224.777,E2 27224.777} C_VEL
LIN {X 0,Y 607.274,Z 780.914,A -85,B 0,C 180,E1 27221.42,E2 27221.42} C_VEL
LIN {X 0,Y 610.139,Z 745.059,A -85,B 0,C 180,E1 27218.331,E2 27218.331} C_VEL
LIN {X 0,Y 612.929,Z 710.531,A -85,B 0,C 180,E1 27215.274,E2 27215.274} C_VEL
LIN {X 0,Y 615.033,Z 683.125,A -85,B 0,C 180,E1 27212.777,E2 27212.777} C_VEL
LIN {X 0,Y 606.577,Z 662.873,A -85,B 0,C 180,E1 27209.856,E2 27209.856} C_VEL
LIN {X 0,Y 598.064,Z 643.41,A -85,B 0,C 180,E1 27206.834,E2 27206.834} C_VEL
LIN {X 0,Y 590.803,Z 627.43,A -85,B 0,C 180,E1 27204.178,E2 27204.178} C_VEL
LIN {X 0,Y 586.677,Z 618.717,A -85,B 0,C 180,E1 27202.655,E2 27202.655} C_VEL
LIN {X 0,Y 585.246,Z 615.08,A -85,B 0,C 180,E1 27202.025,E2 27202.025} C_VEL
LIN {X 0,Y 585.243,Z 615.076,A -85,B 0,C 180,E1 27198.831,E2 27198.831} C_VEL
LIN {X 0,Y 585.242,Z 615.081,A -85,B 0,C 180,E1 27195.661,E2 27195.661} C_VEL
LIN {X 0,Y 585.241,Z 615.078,A -85,B 0,C 180,E1 27192.532,E2 27192.532} C_VEL
LIN {X 0,Y 585.242,Z 615.08,A -85,B 0,C 180,E1 27189.341,E2 27189.341} C_VEL
LIN {X 0,Y 585.242,Z 615.073,A -85,B 0,C 180,E1 27186.179,E2 27186.179} C_VEL
LIN {X 0,Y 585.244,Z 615.078,A -85,B 0,C 180,E1 27182.938,E2 27182.938} C_VEL
LIN {X 0,Y 585.248,Z 615.079,A -85,B 0,C 180,E1 27179.706,E2 27179.706} C_VEL
LIN {X 0,Y 585.253,Z 615.078,A -85,B 0,C 180,E1 27176.376,E2 27176.376} C_VEL
LIN {X 0,Y 585.26,Z 615.075,A -85,B 0,C 180,E1 27173.013,E2 27173.013} C_VEL
LIN {X 0,Y 585.246,Z 615.075,A -85,B 0,C 180,E1 27169.754,E2 27169.754} C_VEL
LIN {X 0,Y 585.255,Z 615.074,A -85,B 0,C 180,E1 27166.464,E2 27166.464} C_VEL
LIN {X 0,Y 585.242,Z 615.076,A -85,B 0,C 180,E1 27163.32,E2 27163.32} C_VEL
LIN {X 0,Y 585.253,Z 615.076,A -85,B 0,C 180,E1 27160.124,E2 27160.124} C_VEL
LIN {X 0,Y 585.244,Z 615.079,A -85,B 0,C 180,E1 27156.968,E2 27156.968} C_VEL
LIN {X 0,Y 585.251,Z 615.081,A -85,B 0,C 180,E1 27153.737,E2 27153.737} C_VEL
LIN {X 0,Y 585.253,Z 615.082,A -85,B 0,C 180,E1 27150.525,E2 27150.525} C_VEL
LIN {X 0,Y 585.258,Z 615.081,A -85,B 0,C 180,E1 27147.196,E2 27147.196} C_VEL
LIN {X 0,Y 585.251,Z 615.079,A -85,B 0,C 180,E1 27143.883,E2 27143.883} C_VEL
LIN {X 0,Y 585.261,Z 615.076,A -85,B 0,C 180,E1 27140.666,E2 27140.666} C_VEL
LIN {X 0,Y 585.245,Z 615.059,A -85,B 0,C 180,E1 27137.42,E2 27137.42} C_VEL
LIN {X 0,Y 585.258,Z 615.081,A -85,B 0,C 180,E1 27134.147,E2 27134.147} C_VEL
LIN {X 0,Y 585.249,Z 615.068,A -85,B 0,C 180,E1 27130.811,E2 27130.811} C_VEL
LIN {X 0,Y 585.258,Z 615.065,A -85,B 0,C 180,E1 27127.458,E2 27127.458} C_VEL
LIN {X 0,Y 585.278,Z 615.239,A -85,B 0,C 180,E1 27124.303,E2 27124.303} C_VEL
LIN {X 0,Y 593.67,Z 640.76,A -85,B 0,C 180,E1 27122.093,E2 27122.093} C_VEL
LIN {X 0,Y 596.165,Z 649.862,A -85,B 0,C 180,E1 27121.326,E2 27121.326} C_VEL
LIN {X 0,Y 594.945,Z 694.705,A -85,B 0,C 180,E1 27118.179,E2 27118.179} C_VEL
LIN {X 0,Y 594.571,Z 705.297,A -85,B 0,C 180,E1 27117.423,E2 27117.423} C_VEL
LIN {X 0,Y 593.451,Z 711.688,A -85,B 0,C 180,E1 27117.011,E2 27117.011} C_VEL
LIN {X 0,Y 587.03,Z 729.292,A -85,B 0,C 180,E1 27116.033,E2 27116.033} C_VEL
LIN {X 0,Y 586.145,Z 734.769,A -85,B 0,C 180,E1 27115.672,E2 27115.672} C_VEL
LIN {X 0,Y 584.559,Z 780.507,A -85,B 0,C 180,E1 27112.421,E2 27112.421} C_VEL
LIN {X 0,Y 583.32,Z 827.275,A -85,B 0,C 180,E1 27109.213,E2 27109.213} C_VEL
LIN {X 0,Y 583.113,Z 842.332,A -85,B 0,C 180,E1 27108.244,E2 27108.244} C_VEL
LIN {X 0,Y 583.884,Z 850.649,A -85,B 0,C 180,E1 27108.111,E2 27108.111} C_VEL
LIN {X 0,Y 582.364,Z 1011.969,A -85,B 0,C 180,E1 27106.078,E2 27106.078} C_VEL
LIN {X 0,Y 582.135,Z 1029.461,A -85,B 0,C 180,E1 27105.676,E2 27105.676} C_VEL
LIN {X 0,Y 581.695,Z 1046.344,A -85,B 0,C 180,E1 27105.093,E2 27105.093} C_VEL
LIN {X 0,Y 581.12,Z 1062.477,A -85,B 0,C 180,E1 27104.344,E2 27104.344} C_VEL
LIN {X 0,Y 580.453,Z 1077.582,A -85,B 0,C 180,E1 27103.446,E2 27103.446} C_VEL
LIN {X 0,Y 579.73,Z 1091.597,A -85,B 0,C 180,E1 27102.398,E2 27102.398} C_VEL
LIN {X 0,Y 579.012,Z 1104.362,A -85,B 0,C 180,E1 27101.222,E2 27101.222} C_VEL
LIN {X 0,Y 578.306,Z 1116.457,A -85,B 0,C 180,E1 27099.854,E2 27099.854} C_VEL
LIN {X 0,Y 577.733,Z 1126.447,A -85,B 0,C 180,E1 27098.458,E2 27098.458} C_VEL
LIN {X 0,Y 577.231,Z 1135.487,A -85,B 0,C 180,E1 27096.863,E2 27096.863} C_VEL
LIN {X 0,Y 576.88,Z 1142.904,A -85,B 0,C 180,E1 27095.17,E2 27095.17} C_VEL
LIN {X 0,Y 576.658,Z 1148.318,A -85,B 0,C 180,E1 27093.478,E2 27093.478} C_VEL
LIN {X 0,Y 576.514,Z 1152.042,A -85,B 0,C 180,E1 27091.688,E2 27091.688} C_VEL
LIN {X 0,Y 576.466,Z 1153.936,A -85,B 0,C 180,E1 27089.899,E2 27089.899} C_VEL
LIN {X 0,Y 576.461,Z 1154.021,A -85,B 0,C 180,E1 27088.11,E2 27088.11} C_VEL
LIN {X 0,Y 576.515,Z 1152.244,A -85,B 0,C 180,E1 27086.319,E2 27086.319} C_VEL
LIN {X 0,Y 576.652,Z 1148.626,A -85,B 0,C 180,E1 27084.526,E2 27084.526} C_VEL
LIN {X 0,Y 576.885,Z 1143.371,A -85,B 0,C 180,E1 27082.83,E2 27082.83} C_VEL
LIN {X 0,Y 577.209,Z 1136.562,A -85,B 0,C 180,E1 27081.23,E2 27081.23} C_VEL
LIN {X 0,Y 577.694,Z 1127.744,A -85,B 0,C 180,E1 27079.629,E2 27079.629} C_VEL
LIN {X 0,Y 578.268,Z 1118.066,A -85,B 0,C 180,E1 27078.226,E2 27078.226} C_VEL
LIN {X 0,Y 578.936,Z 1106.998,A -85,B 0,C 180,E1 27076.922,E2 27076.922} C_VEL
LIN {X 0,Y 579.683,Z 1093.849,A -85,B 0,C 180,E1 27075.668,E2 27075.668} C_VEL
LIN {X 0,Y 580.449,Z 1079.562,A -85,B 0,C 180,E1 27074.564,E2 27074.564} C_VEL
LIN {X 0,Y 581.132,Z 1064.996,A -85,B 0,C 180,E1 27073.66,E2 27073.66} C_VEL
LIN {X 0,Y 581.711,Z 1049.433,A -85,B 0,C 180,E1 27072.906,E2 27072.906} C_VEL
LIN {X 0,Y 582.187,Z 1032.225,A -85,B 0,C 180,E1 27072.281,E2 27072.281} C_VEL
LIN {X 0,Y 582.468,Z 1014.66,A -85,B 0,C 180,E1 27071.842,E2 27071.842} C_VEL
LIN {X 0,Y 582.668,Z 986.621,A -85,B 0,C 180,E1 27071.452,E2 27071.452} C_VEL
LIN {X 0,Y 583.843,Z 846.638,A -85,B 0,C 180,E1 27069.698,E2 27069.698} C_VEL
LIN {X 0,Y 583.194,Z 841.353,A -85,B 0,C 180,E1 27069.579,E2 27069.579} C_VEL
LIN {X 0,Y 584.319,Z 795.245,A -85,B 0,C 180,E1 27066.455,E2 27066.455} C_VEL
LIN {X 0,Y 585.877,Z 749.602,A -85,B 0,C 180,E1 27063.22,E2 27063.22} C_VEL
LIN {X 0,Y 587.519,Z 705.148,A -85,B 0,C 180,E1 27060.027,E2 27060.027} C_VEL
LIN {X 0,Y 588.875,Z 664.82,A -85,B 0,C 180,E1 27057.151,E2 27057.151} C_VEL
LIN {X 0,Y 589.185,Z 652.183,A -85,B 0,C 180,E1 27056.26,E2 27056.26} C_VEL
LIN {X 0,Y 581.813,Z 629.018,A -85,B 0,C 180,E1 27054.211,E2 27054.211} C_VEL
LIN {X 0,Y 577.32,Z 616.052,A -85,B 0,C 180,E1 27053.027,E2 27053.027} C_VEL
LIN {X 0,Y 577.305,Z 616.046,A -85,B 0,C 180,E1 27049.756,E2 27049.756} C_VEL
LIN {X 0,Y 577.313,Z 616.064,A -85,B 0,C 180,E1 27046.527,E2 27046.527} C_VEL
LIN {X 0,Y 577.317,Z 616.068,A -85,B 0,C 180,E1 27043.167,E2 27043.167} C_VEL
LIN {X 0,Y 577.323,Z 616.068,A -85,B 0,C 180,E1 27039.853,E2 27039.853} C_VEL
LIN {X 0,Y 577.356,Z 616.303,A -85,B 0,C 180,E1 27037.632,E2 27037.632} C_VEL
LIN {X 0,Y 578.561,Z 619.456,A -85,B 0,C 180,E1 27037.181,E2 27037.181} C_VEL
LIN {X 0,Y 581.828,Z 626.768,A -85,B 0,C 180,E1 27036.147,E2 27036.147} C_VEL
LIN {X 0,Y 599.292,Z 652.347,A -85,B 0,C 180,E1 27034.342,E2 27034.342} C_VEL
LIN {X 0,Y 604.875,Z 661.168,A -85,B 0,C 180,E1 27033.779,E2 27033.779} C_VEL
LIN {X 0,Y 598.002,Z 900.349,A -85,B 0,C 180,E1 27030.329,E2 27030.329} C_VEL
LIN {X 0,Y 596.55,Z 960.066,A -85,B 0,C 180,E1 27029.462,E2 27029.462} C_VEL
LIN {X 0,Y 595.589,Z 983.233,A -85,B 0,C 180,E1 27028.942,E2 27028.942} C_VEL
LIN {X 0,Y 594.342,Z 1006.474,A -85,B 0,C 180,E1 27028.24,E2 27028.24} C_VEL
LIN {X 0,Y 593,Z 1026.849,A -85,B 0,C 180,E1 27027.462,E2 27027.462} C_VEL
LIN {X 0,Y 591.275,Z 1048.24,A -85,B 0,C 180,E1 27026.462,E2 27026.462} C_VEL
LIN {X 0,Y 589.563,Z 1068.124,A -85,B 0,C 180,E1 27025.356,E2 27025.356} C_VEL
LIN {X 0,Y 587.713,Z 1087.109,A -85,B 0,C 180,E1 27024.099,E2 27024.099} C_VEL
LIN {X 0,Y 585.695,Z 1106.714,A -85,B 0,C 180,E1 27022.589,E2 27022.589} C_VEL
LIN {X 0,Y 583.917,Z 1123.87,A -85,B 0,C 180,E1 27021.051,E2 27021.051} C_VEL
LIN {X 0,Y 582.169,Z 1140.107,A -85,B 0,C 180,E1 27019.359,E2 27019.359} C_VEL
LIN {X 0,Y 580.632,Z 1155.305,A -85,B 0,C 180,E1 27017.54,E2 27017.54} C_VEL
LIN {X 0,Y 579.272,Z 1169.014,A -85,B 0,C 180,E1 27015.621,E2 27015.621} C_VEL
LIN {X 0,Y 578.126,Z 1181.976,A -85,B 0,C 180,E1 27013.503,E2 27013.503} C_VEL
LIN {X 0,Y 577.241,Z 1193.418,A -85,B 0,C 180,E1 27011.288,E2 27011.288} C_VEL
LIN {X 0,Y 576.644,Z 1202.786,A -85,B 0,C 180,E1 27009.079,E2 27009.079} C_VEL
LIN {X 0,Y 576.273,Z 1210.385,A -85,B 0,C 180,E1 27006.876,E2 27006.876} C_VEL
LIN {X 0,Y 576.064,Z 1216.365,A -85,B 0,C 180,E1 27004.679,E2 27004.679} C_VEL
LIN {X 0,Y 575.956,Z 1221.256,A -85,B 0,C 180,E1 27002.189,E2 27002.189} C_VEL
LIN {X 0,Y 575.94,Z 1223.847,A -85,B 0,C 180,E1 27000.099,E2 27000.099} C_VEL
LIN {X 0,Y 575.926,Z 1225.11,A -85,B 0,C 180,E1 26998.11,E2 26998.11} C_VEL
LIN {X 0,Y 575.925,Z 1225.227,A -85,B 0,C 180,E1 26996.217,E2 26996.217} C_VEL
LIN {X 0,Y 575.932,Z 1224.294,A -85,B 0,C 180,E1 26994.321,E2 26994.321} C_VEL
LIN {X 0,Y 575.955,Z 1222.005,A -85,B 0,C 180,E1 26992.217,E2 26992.217} C_VEL
LIN {X 0,Y 576.03,Z 1217.962,A -85,B 0,C 180,E1 26989.903,E2 26989.903} C_VEL
LIN {X 0,Y 576.23,Z 1211.812,A -85,B 0,C 180,E1 26987.473,E2 26987.473} C_VEL
LIN {X 0,Y 576.595,Z 1204.025,A -85,B 0,C 180,E1 26985.128,E2 26985.128} C_VEL
LIN {X 0,Y 577.185,Z 1194.699,A -85,B 0,C 180,E1 26982.872,E2 26982.872} C_VEL
LIN {X 0,Y 577.956,Z 1184.26,A -85,B 0,C 180,E1 26980.809,E2 26980.809} C_VEL
LIN {X 0,Y 578.953,Z 1172.613,A -85,B 0,C 180,E1 26978.841,E2 26978.841} C_VEL
LIN {X 0,Y 580.06,Z 1160.311,A -85,B 0,C 180,E1 26977.072,E2 26977.072} C_VEL
LIN {X 0,Y 581.51,Z 1145.175,A -85,B 0,C 180,E1 26975.194,E2 26975.194} C_VEL
LIN {X 0,Y 582.913,Z 1130.493,A -85,B 0,C 180,E1 26973.623,E2 26973.623} C_VEL
LIN {X 0,Y 584.532,Z 1113.373,A -85,B 0,C 180,E1 26972.05,E2 26972.05} C_VEL
LIN {X 0,Y 586.11,Z 1095.944,A -85,B 0,C 180,E1 26970.664,E2 26970.664} C_VEL
LIN {X 0,Y 587.606,Z 1077.352,A -85,B 0,C 180,E1 26969.417,E2 26969.417} C_VEL
LIN {X 0,Y 589.112,Z 1056.771,A -85,B 0,C 180,E1 26968.25,E2 26968.25} C_VEL
LIN {X 0,Y 590.23,Z 1038.176,A -85,B 0,C 180,E1 26967.372,E2 26967.372} C_VEL
LIN {X 0,Y 591.272,Z 1016.538,A -85,B 0,C 180,E1 26966.544,E2 26966.544} C_VEL
LIN {X 0,Y 592.026,Z 995.161,A -85,B 0,C 180,E1 26965.901,E2 26965.901} C_VEL
LIN {X 0,Y 592.478,Z 973.457,A -85,B 0,C 180,E1 26965.435,E2 26965.435} C_VEL
LIN {X 0,Y 592.684,Z 945.634,A -85,B 0,C 180,E1 26965.048,E2 26965.048} C_VEL
LIN {X 0,Y 594.015,Z 815.429,A -85,B 0,C 180,E1 26963.479,E2 26963.479} C_VEL
LIN {X 0,Y 595.892,Z 706.592,A -85,B 0,C 180,E1 26962.003,E2 26962.003} C_VEL
LIN {X 0,Y 596.727,Z 674.931,A -85,B 0,C 180,E1 26961.532,E2 26961.532} C_VEL
LIN {X 0,Y 598.102,Z 674.302,A -85,B 0,C 180,E1 26961.369,E2 26961.369} C_VEL
LIN {X 0,Y 592.405,Z 684.217,A -85,B 0,C 180,E1 26960.022,E2 26960.022} C_VEL
LIN {X 0,Y 587.752,Z 696.462,A -85,B 0,C 180,E1 26958.612,E2 26958.612} C_VEL
LIN {X 0,Y 584.215,Z 710.693,A -85,B 0,C 180,E1 26957.198,E2 26957.198} C_VEL
LIN {X 0,Y 581.471,Z 728.372,A -85,B 0,C 180,E1 26955.673,E2 26955.673} C_VEL
LIN {X 0,Y 579.312,Z 752.1,A -85,B 0,C 180,E1 26953.868,E2 26953.868} C_VEL
LIN {X 0,Y 578.426,Z 780.483,A -85,B 0,C 180,E1 26951.896,E2 26951.896} C_VEL
LIN {X 0,Y 579.812,Z 802.287,A -85,B 0,C 180,E1 26950.423,E2 26950.423} C_VEL
LIN {X 0,Y 583.129,Z 821.613,A -85,B 0,C 180,E1 26949.126,E2 26949.126} C_VEL
LIN {X 0,Y 588.183,Z 838.705,A -85,B 0,C 180,E1 26947.981,E2 26947.981} C_VEL
LIN {X 0,Y 595.472,Z 855.584,A -85,B 0,C 180,E1 26946.858,E2 26946.858} C_VEL
LIN {X 0,Y 604.1,Z 870.495,A -85,B 0,C 180,E1 26945.883,E2 26945.883} C_VEL
LIN {X 0,Y 614.121,Z 884.034,A -85,B 0,C 180,E1 26945.018,E2 26945.018} C_VEL
LIN {X 0,Y 626.268,Z 897.163,A -85,B 0,C 180,E1 26944.205,E2 26944.205} C_VEL
LIN {X 0,Y 627.397,Z 898.491,A -85,B 0,C 180,E1 26944.125,E2 26944.125} C_VEL
LIN {X 0,Y 616.405,Z 910.814,A -85,B 0,C 180,E1 26943.473,E2 26943.473} C_VEL
LIN {X 0,Y 607.628,Z 923.383,A -85,B 0,C 180,E1 26942.779,E2 26942.779} C_VEL
LIN {X 0,Y 602.635,Z 931.524,A -85,B 0,C 180,E1 26942.345,E2 26942.345} C_VEL
LIN {X 0,Y 597.417,Z 947.381,A -85,B 0,C 180,E1 26942.338,E2 26942.338} C_VEL
LIN {X 0,Y 593.666,Z 962.602,A -85,B 0,C 180,E1 26942.29,E2 26942.29} C_VEL
LIN {X 0,Y 592.183,Z 975.415,A -85,B 0,C 180,E1 26942.154,E2 26942.154} C_VEL
LIN {X 0,Y 591.099,Z 1006.857,A -85,B 0,C 180,E1 26941.571,E2 26941.571} C_VEL
LIN {X 0,Y 589.743,Z 1036.155,A -85,B 0,C 180,E1 26940.851,E2 26940.851} C_VEL
LIN {X 0,Y 588.41,Z 1064.198,A -85,B 0,C 180,E1 26939.974,E2 26939.974} C_VEL
LIN {X 0,Y 587.081,Z 1091.397,A -85,B 0,C 180,E1 26938.928,E2 26938.928} C_VEL
LIN {X 0,Y 585.798,Z 1116.326,A -85,B 0,C 180,E1 26937.775,E2 26937.775} C_VEL
LIN {X 0,Y 584.509,Z 1139.364,A -85,B 0,C 180,E1 26936.519,E2 26936.519} C_VEL
LIN {X 0,Y 583.217,Z 1161.311,A -85,B 0,C 180,E1 26935.119,E2 26935.119} C_VEL
LIN {X 0,Y 581.881,Z 1182.277,A -85,B 0,C 180,E1 26933.549,E2 26933.549} C_VEL
LIN {X 0,Y 580.735,Z 1200.145,A -85,B 0,C 180,E1 26931.994,E2 26931.994} C_VEL
LIN {X 0,Y 579.63,Z 1216.923,A -85,B 0,C 180,E1 26930.289,E2 26930.289} C_VEL
LIN {X 0,Y 578.722,Z 1230.9,A -85,B 0,C 180,E1 26928.642,E2 26928.642} C_VEL
LIN {X 0,Y 577.92,Z 1243.637,A -85,B 0,C 180,E1 26926.899,E2 26926.899} C_VEL
LIN {X 0,Y 577.208,Z 1256.298,A -85,B 0,C 180,E1 26924.845,E2 26924.845} C_VEL
LIN {X 0,Y 576.706,Z 1265.773,A -85,B 0,C 180,E1 26922.993,E2 26922.993} C_VEL
LIN {X 0,Y 576.41,Z 1272.701,A -85,B 0,C 180,E1 26921.407,E2 26921.407} C_VEL
LIN {X 0,Y 576.191,Z 1278.983,A -85,B 0,C 180,E1 26919.692,E2 26919.692} C_VEL
LIN {X 0,Y 576.034,Z 1284.104,A -85,B 0,C 180,E1 26917.983,E2 26917.983} C_VEL
LIN {X 0,Y 575.97,Z 1288.349,A -85,B 0,C 180,E1 26916.18,E2 26916.18} C_VEL
LIN {X 0,Y 575.921,Z 1291.46,A -85,B 0,C 180,E1 26914.382,E2 26914.382} C_VEL
LIN {X 0,Y 575.904,Z 1293.49,A -85,B 0,C 180,E1 26912.589,E2 26912.589} C_VEL
LIN {X 0,Y 575.907,Z 1294.474,A -85,B 0,C 180,E1 26910.797,E2 26910.797} C_VEL
LIN {X 0,Y 575.915,Z 1294.424,A -85,B 0,C 180,E1 26909.007,E2 26909.007} C_VEL
LIN {X 0,Y 575.911,Z 1293.267,A -85,B 0,C 180,E1 26907.115,E2 26907.115} C_VEL
LIN {X 0,Y 575.924,Z 1290.818,A -85,B 0,C 180,E1 26905.121,E2 26905.121} C_VEL
LIN {X 0,Y 576.004,Z 1286.162,A -85,B 0,C 180,E1 26902.721,E2 26902.721} C_VEL
LIN {X 0,Y 576.141,Z 1280.349,A -85,B 0,C 180,E1 26900.613,E2 26900.613} C_VEL
LIN {X 0,Y 576.376,Z 1273.739,A -85,B 0,C 180,E1 26898.697,E2 26898.697} C_VEL
LIN {X 0,Y 576.725,Z 1266.183,A -85,B 0,C 180,E1 26896.874,E2 26896.874} C_VEL
LIN {X 0,Y 577.264,Z 1256.742,A -85,B 0,C 180,E1 26894.942,E2 26894.942} C_VEL
LIN {X 0,Y 578.134,Z 1243.633,A -85,B 0,C 180,E1 26892.688,E2 26892.688} C_VEL
LIN {X 0,Y 579.14,Z 1230.262,A -85,B 0,C 180,E1 26890.747,E2 26890.747} C_VEL
LIN {X 0,Y 580.361,Z 1215.613,A -85,B 0,C 180,E1 26888.897,E2 26888.897} C_VEL
LIN {X 0,Y 582.005,Z 1197.153,A -85,B 0,C 180,E1 26886.885,E2 26886.885} C_VEL
LIN {X 0,Y 583.754,Z 1178.369,A -85,B 0,C 180,E1 26885.135,E2 26885.135} C_VEL
LIN {X 0,Y 585.495,Z 1159.96,A -85,B 0,C 180,E1 26883.641,E2 26883.641} C_VEL
LIN {X 0,Y 587.624,Z 1137.998,A -85,B 0,C 180,E1 26882.102,E2 26882.102} C_VEL
LIN {X 0,Y 589.548,Z 1117.612,A -85,B 0,C 180,E1 26880.874,E2 26880.874} C_VEL
LIN {X 0,Y 591.794,Z 1093.711,A -85,B 0,C 180,E1 26879.658,E2 26879.658} C_VEL
LIN {X 0,Y 593.549,Z 1073.738,A -85,B 0,C 180,E1 26878.803,E2 26878.803} C_VEL
LIN {X 0,Y 595.683,Z 1048.163,A -85,B 0,C 180,E1 26877.911,E2 26877.911} C_VEL
LIN {X 0,Y 597.321,Z 1026.531,A -85,B 0,C 180,E1 26877.321,E2 26877.321} C_VEL
LIN {X 0,Y 598.888,Z 1000.49,A -85,B 0,C 180,E1 26876.795,E2 26876.795} C_VEL
LIN {X 0,Y 600.185,Z 971.114,A -85,B 0,C 180,E1 26876.363,E2 26876.363} C_VEL
LIN {X 0,Y 601.86,Z 958.854,A -85,B 0,C 180,E1 26876.242,E2 26876.242} C_VEL
LIN {X 0,Y 608.616,Z 946.51,A -85,B 0,C 180,E1 26875.589,E2 26875.589} C_VEL
LIN {X 0,Y 619.277,Z 929.618,A -85,B 0,C 180,E1 26874.785,E2 26874.785} C_VEL
LIN {X 0,Y 629.495,Z 916.3,A -85,B 0,C 180,E1 26874.26,E2 26874.26} C_VEL
LIN {X 0,Y 632.62,Z 912.417,A -85,B 0,C 180,E1 26874.117,E2 26874.117} C_VEL
LIN {X 0,Y 622.221,Z 903.164,A -85,B 0,C 180,E1 26872.829,E2 26872.829} C_VEL
LIN {X 0,Y 613.689,Z 892.801,A -85,B 0,C 180,E1 26871.511,E2 26871.511} C_VEL
LIN {X 0,Y 606.923,Z 881.198,A -85,B 0,C 180,E1 26870.146,E2 26870.146} C_VEL
LIN {X 0,Y 601.686,Z 867.796,A -85,B 0,C 180,E1 26868.69,E2 26868.69} C_VEL
LIN {X 0,Y 598.463,Z 853.548,A -85,B 0,C 180,E1 26867.249,E2 26867.249} C_VEL
LIN {X 0,Y 597.036,Z 837.021,A -85,B 0,C 180,E1 26865.706,E2 26865.706} C_VEL
LIN {X 0,Y 597.669,Z 817.11,A -85,B 0,C 180,E1 26863.971,E2 26863.971} C_VEL
LIN {X 0,Y 600.67,Z 779.974,A -85,B 0,C 180,E1 26860.817,E2 26860.817} C_VEL
LIN {X 0,Y 603.581,Z 745.268,A -85,B 0,C 180,E1 26857.799,E2 26857.799} C_VEL
LIN {X 0,Y 606.441,Z 711.524,A -85,B 0,C 180,E1 26854.784,E2 26854.784} C_VEL
LIN {X 0,Y 608.367,Z 686.933,A -85,B 0,C 180,E1 26852.51,E2 26852.51} C_VEL
LIN {X 0,Y 599.93,Z 666.719,A -85,B 0,C 180,E1 26849.56,E2 26849.56} C_VEL
LIN {X 0,Y 591.842,Z 648.18,A -85,B 0,C 180,E1 26846.66,E2 26846.66} C_VEL
LIN {X 0,Y 584.694,Z 632.407,A -85,B 0,C 180,E1 26844.017,E2 26844.017} C_VEL
LIN {X 0,Y 580.314,Z 623.224,A -85,B 0,C 180,E1 26842.383,E2 26842.383} C_VEL
LIN {X 0,Y 578.576,Z 619.503,A -85,B 0,C 180,E1 26841.705,E2 26841.705} C_VEL
LIN {X 0,Y 577.322,Z 616.064,A -85,B 0,C 180,E1 26841.115,E2 26841.115} C_VEL
LIN {X 0,Y 577.311,Z 616.07,A -85,B 0,C 180,E1 26837.852,E2 26837.852} C_VEL
LIN {X 0,Y 577.317,Z 616.066,A -85,B 0,C 180,E1 26834.545,E2 26834.545} C_VEL
LIN {X 0,Y 577.308,Z 616.065,A -85,B 0,C 180,E1 26831.287,E2 26831.287} C_VEL
LIN {X 0,Y 577.323,Z 616.065,A -85,B 0,C 180,E1 26827.964,E2 26827.964} C_VEL
LIN {X 0,Y 577.313,Z 616.067,A -85,B 0,C 180,E1 26824.57,E2 26824.57} C_VEL
LIN {X 0,Y 577.308,Z 616.063,A -85,B 0,C 180,E1 26821.29,E2 26821.29} C_VEL
LIN {X 0,Y 577.306,Z 616.063,A -85,B 0,C 180,E1 26818.114,E2 26818.114} C_VEL
LIN {X 0,Y 577.303,Z 616.067,A -85,B 0,C 180,E1 26814.833,E2 26814.833} C_VEL
LIN {X 0,Y 577.304,Z 616.068,A -85,B 0,C 180,E1 26811.634,E2 26811.634} C_VEL
LIN {X 0,Y 577.305,Z 616.068,A -85,B 0,C 180,E1 26808.41,E2 26808.41} C_VEL
LIN {X 0,Y 577.313,Z 616.068,A -85,B 0,C 180,E1 26805.106,E2 26805.106} C_VEL
LIN {X 0,Y 577.319,Z 616.069,A -85,B 0,C 180,E1 26801.731,E2 26801.731} C_VEL
LIN {X 0,Y 577.327,Z 616.069,A -85,B 0,C 180,E1 26798.352,E2 26798.352} C_VEL
LIN {X 0,Y 577.322,Z 616.07,A -85,B 0,C 180,E1 26795.001,E2 26795.001} C_VEL
LIN {X 0,Y 577.317,Z 616.069,A -85,B 0,C 180,E1 26791.618,E2 26791.618} C_VEL
LIN {X 0,Y 577.321,Z 616.065,A -85,B 0,C 180,E1 26788.23,E2 26788.23} C_VEL
LIN {X 0,Y 577.309,Z 616.06,A -85,B 0,C 180,E1 26784.899,E2 26784.899} C_VEL
LIN {X 0,Y 577.305,Z 616.061,A -85,B 0,C 180,E1 26781.68,E2 26781.68} C_VEL
LIN {X 0,Y 577.305,Z 616.064,A -85,B 0,C 180,E1 26778.443,E2 26778.443} C_VEL
LIN {X 0,Y 577.306,Z 616.061,A -85,B 0,C 180,E1 26775.176,E2 26775.176} C_VEL
LIN {X 0,Y 577.304,Z 616.051,A -85,B 0,C 180,E1 26771.953,E2 26771.953} C_VEL
LIN {X 0,Y 577.312,Z 616.07,A -85,B 0,C 180,E1 26768.698,E2 26768.698} C_VEL
LIN {X 0,Y 577.321,Z 616.067,A -85,B 0,C 180,E1 26765.338,E2 26765.338} C_VEL
LIN {X 0,Y 577.315,Z 616.078,A -85,B 0,C 180,E1 26764.697,E2 26764.697} C_VEL
LIN {X 0,Y 586.274,Z 643.163,A -85,B 0,C 180,E1 26762.319,E2 26762.319} C_VEL
LIN {X 0,Y 588.815,Z 652.359,A -85,B 0,C 180,E1 26761.533,E2 26761.533} C_VEL
LIN {X 0,Y 587.574,Z 695.163,A -85,B 0,C 180,E1 26758.509,E2 26758.509} C_VEL
LIN {X 0,Y 586.145,Z 734.769,A -85,B 0,C 180,E1 26755.672,E2 26755.672} C_VEL
LIN {X 0,Y 585.017,Z 741.177,A -85,B 0,C 180,E1 26755.256,E2 26755.256} C_VEL
LIN {X 0,Y 578.591,Z 758.804,A -85,B 0,C 180,E1 26754.27,E2 26754.27} C_VEL
LIN {X 0,Y 577.684,Z 764.311,A -85,B 0,C 180,E1 26753.909,E2 26753.909} C_VEL
LIN {X 0,Y 576.169,Z 812.768,A -85,B 0,C 180,E1 26750.519,E2 26750.519} C_VEL
LIN {X 0,Y 575.578,Z 843.224,A -85,B 0,C 180,E1 26748.501,E2 26748.501} C_VEL
LIN {X 0,Y 576.339,Z 851.393,A -85,B 0,C 180,E1 26748.367,E2 26748.367} C_VEL
LIN {X 0,Y 574.738,Z 1012.858,A -85,B 0,C 180,E1 26746.307,E2 26746.307} C_VEL
LIN {X 0,Y 574.505,Z 1030.314,A -85,B 0,C 180,E1 26745.901,E2 26745.901} C_VEL
LIN {X 0,Y 574.085,Z 1046.287,A -85,B 0,C 180,E1 26745.35,E2 26745.35} C_VEL
LIN {X 0,Y 573.483,Z 1062.635,A -85,B 0,C 180,E1 26744.591,E2 26744.591} C_VEL
LIN {X 0,Y 572.781,Z 1077.894,A -85,B 0,C 180,E1 26743.681,E2 26743.681} C_VEL
LIN {X 0,Y 572.026,Z 1092.069,A -85,B 0,C 180,E1 26742.619,E2 26742.619} C_VEL
LIN {X 0,Y 571.25,Z 1105.123,A -85,B 0,C 180,E1 26741.406,E2 26741.406} C_VEL
LIN {X 0,Y 570.537,Z 1116.673,A -85,B 0,C 180,E1 26740.092,E2 26740.092} C_VEL
LIN {X 0,Y 569.919,Z 1126.803,A -85,B 0,C 180,E1 26738.677,E2 26738.677} C_VEL
LIN {X 0,Y 569.411,Z 1135.498,A -85,B 0,C 180,E1 26737.161,E2 26737.161} C_VEL
LIN {X 0,Y 569.024,Z 1142.729,A -85,B 0,C 180,E1 26735.545,E2 26735.545} C_VEL
LIN {X 0,Y 568.76,Z 1148.456,A -85,B 0,C 180,E1 26733.829,E2 26733.829} C_VEL
LIN {X 0,Y 568.606,Z 1152.376,A -85,B 0,C 180,E1 26732.115,E2 26732.115} C_VEL
LIN {X 0,Y 568.53,Z 1154.632,A -85,B 0,C 180,E1 26730.301,E2 26730.301} C_VEL
LIN {X 0,Y 568.511,Z 1155.084,A -85,B 0,C 180,E1 26728.487,E2 26728.487} C_VEL
LIN {X 0,Y 568.564,Z 1153.758,A -85,B 0,C 180,E1 26726.672,E2 26726.672} C_VEL
LIN {X 0,Y 568.683,Z 1150.773,A -85,B 0,C 180,E1 26724.955,E2 26724.955} C_VEL
LIN {X 0,Y 568.897,Z 1146.006,A -85,B 0,C 180,E1 26723.236,E2 26723.236} C_VEL
LIN {X 0,Y 569.235,Z 1139.347,A -85,B 0,C 180,E1 26721.514,E2 26721.514} C_VEL
LIN {X 0,Y 569.715,Z 1131.081,A -85,B 0,C 180,E1 26719.891,E2 26719.891} C_VEL
LIN {X 0,Y 570.322,Z 1121.169,A -85,B 0,C 180,E1 26718.367,E2 26718.367} C_VEL
LIN {X 0,Y 571.059,Z 1109.686,A -85,B 0,C 180,E1 26716.945,E2 26716.945} C_VEL
LIN {X 0,Y 571.843,Z 1097.024,A -85,B 0,C 180,E1 26715.674,E2 26715.674} C_VEL
LIN {X 0,Y 572.625,Z 1083.177,A -85,B 0,C 180,E1 26714.554,E2 26714.554} C_VEL
LIN {X 0,Y 573.388,Z 1067.864,A -85,B 0,C 180,E1 26713.559,E2 26713.559} C_VEL
LIN {X 0,Y 574.02,Z 1052.509,A -85,B 0,C 180,E1 26712.774,E2 26712.774} C_VEL
LIN {X 0,Y 574.521,Z 1035.702,A -85,B 0,C 180,E1 26712.129,E2 26712.129} C_VEL
LIN {X 0,Y 574.841,Z 1017.759,A -85,B 0,C 180,E1 26711.651,E2 26711.651} C_VEL
LIN {X 0,Y 574.974,Z 997.861,A -85,B 0,C 180,E1 26711.339,E2 26711.339} C_VEL
LIN {X 0,Y 576.337,Z 847.51,A -85,B 0,C 180,E1 26709.432,E2 26709.432} C_VEL
LIN {X 0,Y 575.684,Z 842.476,A -85,B 0,C 180,E1 26709.327,E2 26709.327} C_VEL
LIN {X 0,Y 576.863,Z 796.222,A -85,B 0,C 180,E1 26706.179,E2 26706.179} C_VEL
LIN {X 0,Y 578.468,Z 751.069,A -85,B 0,C 180,E1 26702.96,E2 26702.96} C_VEL
LIN {X 0,Y 580.195,Z 705.922,A -85,B 0,C 180,E1 26699.702,E2 26699.702} C_VEL
LIN {X 0,Y 581.594,Z 666.216,A -85,B 0,C 180,E1 26696.853,E2 26696.853} C_VEL
LIN {X 0,Y 581.907,Z 654.891,A -85,B 0,C 180,E1 26696.05,E2 26696.05} C_VEL
LIN {X 0,Y 574.498,Z 631.59,A -85,B 0,C 180,E1 26693.964,E2 26693.964} C_VEL
LIN {X 0,Y 569.382,Z 617.046,A -85,B 0,C 180,E1 26692.603,E2 26692.603} C_VEL
LIN {X 0,Y 569.389,Z 617.037,A -85,B 0,C 180,E1 26689.211,E2 26689.211} C_VEL
LIN {X 0,Y 569.367,Z 617.057,A -85,B 0,C 180,E1 26685.912,E2 26685.912} C_VEL
LIN {X 0,Y 569.365,Z 617.054,A -85,B 0,C 180,E1 26682.622,E2 26682.622} C_VEL
LIN {X 0,Y 569.385,Z 617.057,A -85,B 0,C 180,E1 26679.342,E2 26679.342} C_VEL
LIN {X 0,Y 569.4,Z 617.296,A -85,B 0,C 180,E1 26678.372,E2 26678.372} C_VEL
LIN {X 0,Y 570.964,Z 620.921,A -85,B 0,C 180,E1 26677.832,E2 26677.832} C_VEL
LIN {X 0,Y 574.439,Z 628.697,A -85,B 0,C 180,E1 26676.719,E2 26676.719} C_VEL
LIN {X 0,Y 593.931,Z 657.343,A -85,B 0,C 180,E1 26674.652,E2 26674.652} C_VEL
LIN {X 0,Y 598.398,Z 664.534,A -85,B 0,C 180,E1 26674.195,E2 26674.195} C_VEL
LIN {X 0,Y 591.1,Z 902.444,A -85,B 0,C 180,E1 26670.7,E2 26670.7} C_VEL
LIN {X 0,Y 589.577,Z 961.093,A -85,B 0,C 180,E1 26669.831,E2 26669.831} C_VEL
LIN {X 0,Y 588.588,Z 984.007,A -85,B 0,C 180,E1 26669.309,E2 26669.309} C_VEL
LIN {X 0,Y 587.263,Z 1007.669,A -85,B 0,C 180,E1 26668.584,E2 26668.584} C_VEL
LIN {X 0,Y 585.82,Z 1028.551,A -85,B 0,C 180,E1 26667.773,E2 26667.773} C_VEL
LIN {X 0,Y 584.027,Z 1049.72,A -85,B 0,C 180,E1 26666.761,E2 26666.761} C_VEL
LIN {X 0,Y 582.165,Z 1070.149,A -85,B 0,C 180,E1 26665.598,E2 26665.598} C_VEL
LIN {X 0,Y 580.246,Z 1089.078,A -85,B 0,C 180,E1 26664.321,E2 26664.321} C_VEL
LIN {X 0,Y 578.145,Z 1108.454,A -85,B 0,C 180,E1 26662.793,E2 26662.793} C_VEL
LIN {X 0,Y 576.27,Z 1125.777,A -85,B 0,C 180,E1 26661.209,E2 26661.209} C_VEL
LIN {X 0,Y 574.474,Z 1141.563,A -85,B 0,C 180,E1 26659.523,E2 26659.523} C_VEL
LIN {X 0,Y 572.779,Z 1157.36,A -85,B 0,C 180,E1 26657.578,E2 26657.578} C_VEL
LIN {X 0,Y 571.451,Z 1170.241,A -85,B 0,C 180,E1 26655.736,E2 26655.736} C_VEL
LIN {X 0,Y 570.296,Z 1182.508,A -85,B 0,C 180,E1 26653.692,E2 26653.692} C_VEL
LIN {X 0,Y 569.399,Z 1193.493,A -85,B 0,C 180,E1 26651.548,E2 26651.548} C_VEL
LIN {X 0,Y 568.741,Z 1202.923,A -85,B 0,C 180,E1 26649.308,E2 26649.308} C_VEL
LIN {X 0,Y 568.34,Z 1210.632,A -85,B 0,C 180,E1 26647.074,E2 26647.074} C_VEL
LIN {X 0,Y 568.103,Z 1216.641,A -85,B 0,C 180,E1 26644.846,E2 26644.846} C_VEL
LIN {X 0,Y 567.979,Z 1221.609,A -85,B 0,C 180,E1 26642.321,E2 26642.321} C_VEL
LIN {X 0,Y 567.957,Z 1224.378,A -85,B 0,C 180,E1 26640.101,E2 26640.101} C_VEL
LIN {X 0,Y 567.934,Z 1225.684,A -85,B 0,C 180,E1 26637.881,E2 26637.881} C_VEL
LIN {X 0,Y 567.932,Z 1225.625,A -85,B 0,C 180,E1 26635.759,E2 26635.759} C_VEL
LIN {X 0,Y 567.939,Z 1224.07,A -85,B 0,C 180,E1 26633.429,E2 26633.429} C_VEL
LIN {X 0,Y 567.999,Z 1220.869,A -85,B 0,C 180,E1 26631.088,E2 26631.088} C_VEL
LIN {X 0,Y 568.11,Z 1216.442,A -85,B 0,C 180,E1 26628.94,E2 26628.94} C_VEL
LIN {X 0,Y 568.368,Z 1210.306,A -85,B 0,C 180,E1 26626.676,E2 26626.676} C_VEL
LIN {X 0,Y 568.79,Z 1202.463,A -85,B 0,C 180,E1 26624.44,E2 26624.44} C_VEL
LIN {X 0,Y 569.472,Z 1192.856,A -85,B 0,C 180,E1 26622.211,E2 26622.211} C_VEL
LIN {X 0,Y 570.371,Z 1182.09,A -85,B 0,C 180,E1 26620.117,E2 26620.117} C_VEL
LIN {X 0,Y 571.47,Z 1169.767,A -85,B 0,C 180,E1 26618.119,E2 26618.119} C_VEL
LIN {X 0,Y 572.863,Z 1155.624,A -85,B 0,C 180,E1 26616.151,E2 26616.151} C_VEL
LIN {X 0,Y 574.349,Z 1140.9,A -85,B 0,C 180,E1 26614.396,E2 26614.396} C_VEL
LIN {X 0,Y 575.945,Z 1125.003,A -85,B 0,C 180,E1 26612.771,E2 26612.771} C_VEL
LIN {X 0,Y 577.596,Z 1108.112,A -85,B 0,C 180,E1 26611.27,E2 26611.27} C_VEL
LIN {X 0,Y 579.227,Z 1089.88,A -85,B 0,C 180,E1 26609.902,E2 26609.902} C_VEL
LIN {X 0,Y 580.863,Z 1069.941,A -85,B 0,C 180,E1 26608.629,E2 26608.629} C_VEL
LIN {X 0,Y 582.216,Z 1050.741,A -85,B 0,C 180,E1 26607.6,E2 26607.6} C_VEL
LIN {X 0,Y 583.336,Z 1030.995,A -85,B 0,C 180,E1 26606.735,E2 26606.735} C_VEL
LIN {X 0,Y 584.314,Z 1010.04,A -85,B 0,C 180,E1 26605.989,E2 26605.989} C_VEL
LIN {X 0,Y 584.897,Z 989.407,A -85,B 0,C 180,E1 26605.434,E2 26605.434} C_VEL
LIN {X 0,Y 585.247,Z 965.988,A -85,B 0,C 180,E1 26604.987,E2 26604.987} C_VEL
LIN {X 0,Y 586.88,Z 817.843,A -85,B 0,C 180,E1 26603.15,E2 26603.15} C_VEL
LIN {X 0,Y 588.966,Z 713.471,A -85,B 0,C 180,E1 26601.688,E2 26601.688} C_VEL
LIN {X 0,Y 589.814,Z 682.017,A -85,B 0,C 180,E1 26601.206,E2 26601.206} C_VEL
LIN {X 0,Y 589.33,Z 682.029,A -85,B 0,C 180,E1 26601.149,E2 26601.149} C_VEL
LIN {X 0,Y 583.881,Z 692.277,A -85,B 0,C 180,E1 26599.788,E2 26599.788} C_VEL
LIN {X 0,Y 579.399,Z 704.907,A -85,B 0,C 180,E1 26598.353,E2 26598.353} C_VEL
LIN {X 0,Y 575.954,Z 719.939,A -85,B 0,C 180,E1 26596.881,E2 26596.881} C_VEL
LIN {X 0,Y 573.198,Z 739.194,A -85,B 0,C 180,E1 26595.234,E2 26595.234} C_VEL
LIN {X 0,Y 571.12,Z 764.808,A -85,B 0,C 180,E1 26593.293,E2 26593.293} C_VEL
LIN {X 0,Y 571.001,Z 790.876,A -85,B 0,C 180,E1 26591.448,E2 26591.448} C_VEL
LIN {X 0,Y 573.261,Z 812.681,A -85,B 0,C 180,E1 26589.932,E2 26589.932} C_VEL
LIN {X 0,Y 577.387,Z 831.33,A -85,B 0,C 180,E1 26588.646,E2 26588.646} C_VEL
LIN {X 0,Y 583.37,Z 848.337,A -85,B 0,C 180,E1 26587.479,E2 26587.479} C_VEL
LIN {X 0,Y 591.228,Z 864.464,A -85,B 0,C 180,E1 26586.388,E2 26586.388} C_VEL
LIN {X 0,Y 600.883,Z 879.551,A -85,B 0,C 180,E1 26585.387,E2 26585.387} C_VEL
LIN {X 0,Y 611.682,Z 892.908,A -85,B 0,C 180,E1 26584.526,E2 26584.526} C_VEL
LIN {X 0,Y 616.973,Z 898.755,A -85,B 0,C 180,E1 26584.161,E2 26584.161} C_VEL
LIN {X 0,Y 606.713,Z 911.177,A -85,B 0,C 180,E1 26583.497,E2 26583.497} C_VEL
LIN {X 0,Y 596.694,Z 926.722,A -85,B 0,C 180,E1 26582.656,E2 26582.656} C_VEL
LIN {X 0,Y 591.077,Z 943.159,A -85,B 0,C 180,E1 26582.67,E2 26582.67} C_VEL
LIN {X 0,Y 586.665,Z 960.478,A -85,B 0,C 180,E1 26582.62,E2 26582.62} C_VEL
LIN {X 0,Y 584.905,Z 973.662,A -85,B 0,C 180,E1 26582.48,E2 26582.48} C_VEL
LIN {X 0,Y 583.651,Z 1005.044,A -85,B 0,C 180,E1 26581.877,E2 26581.877} C_VEL
LIN {X 0,Y 582.153,Z 1035.04,A -85,B 0,C 180,E1 26581.117,E2 26581.117} C_VEL
LIN {X 0,Y 580.725,Z 1063.111,A -85,B 0,C 180,E1 26580.213,E2 26580.213} C_VEL
LIN {X 0,Y 579.365,Z 1089.585,A -85,B 0,C 180,E1 26579.175,E2 26579.175} C_VEL
LIN {X 0,Y 577.994,Z 1114.86,A -85,B 0,C 180,E1 26577.993,E2 26577.993} C_VEL
LIN {X 0,Y 576.69,Z 1137.898,A -85,B 0,C 180,E1 26576.725,E2 26576.725} C_VEL
LIN {X 0,Y 575.363,Z 1159.914,A -85,B 0,C 180,E1 26575.311,E2 26575.311} C_VEL
LIN {X 0,Y 574,Z 1180.985,A -85,B 0,C 180,E1 26573.729,E2 26573.729} C_VEL
LIN {X 0,Y 572.824,Z 1198.988,A -85,B 0,C 180,E1 26572.151,E2 26572.151} C_VEL
LIN {X 0,Y 571.661,Z 1216.565,A -85,B 0,C 180,E1 26570.361,E2 26570.361} C_VEL
LIN {X 0,Y 570.681,Z 1231.476,A -85,B 0,C 180,E1 26568.578,E2 26568.578} C_VEL
LIN {X 0,Y 569.77,Z 1246.092,A -85,B 0,C 180,E1 26566.518,E2 26566.518} C_VEL
LIN {X 0,Y 569.153,Z 1257.058,A -85,B 0,C 180,E1 26564.655,E2 26564.655} C_VEL
LIN {X 0,Y 568.716,Z 1265.405,A -85,B 0,C 180,E1 26563.007,E2 26563.007} C_VEL
LIN {X 0,Y 568.41,Z 1272.508,A -85,B 0,C 180,E1 26561.364,E2 26561.364} C_VEL
LIN {X 0,Y 568.194,Z 1278.794,A -85,B 0,C 180,E1 26559.625,E2 26559.625} C_VEL
LIN {X 0,Y 568.041,Z 1283.903,A -85,B 0,C 180,E1 26557.893,E2 26557.893} C_VEL
LIN {X 0,Y 567.974,Z 1288.117,A -85,B 0,C 180,E1 26556.065,E2 26556.065} C_VEL
LIN {X 0,Y 567.937,Z 1291.182,A -85,B 0,C 180,E1 26554.242,E2 26554.242} C_VEL
LIN {X 0,Y 567.923,Z 1293.233,A -85,B 0,C 180,E1 26552.322,E2 26552.322} C_VEL
LIN {X 0,Y 567.928,Z 1294.183,A -85,B 0,C 180,E1 26550.102,E2 26550.102} C_VEL
LIN {X 0,Y 567.918,Z 1293.322,A -85,B 0,C 180,E1 26547.681,E2 26547.681} C_VEL
LIN {X 0,Y 567.927,Z 1291.206,A -85,B 0,C 180,E1 26545.66,E2 26545.66} C_VEL
LIN {X 0,Y 567.971,Z 1287.991,A -85,B 0,C 180,E1 26543.735,E2 26543.735} C_VEL
LIN {X 0,Y 568.049,Z 1283.553,A -85,B 0,C 180,E1 26541.804,E2 26541.804} C_VEL
LIN {X 0,Y 568.258,Z 1277.037,A -85,B 0,C 180,E1 26539.611,E2 26539.611} C_VEL
LIN {X 0,Y 568.63,Z 1268.232,A -85,B 0,C 180,E1 26537.304,E2 26537.304} C_VEL
LIN {X 0,Y 569.172,Z 1258.634,A -85,B 0,C 180,E1 26535.244,E2 26535.244} C_VEL
LIN {X 0,Y 569.923,Z 1247.273,A -85,B 0,C 180,E1 26533.175,E2 26533.175} C_VEL
LIN {X 0,Y 571.067,Z 1232.394,A -85,B 0,C 180,E1 26530.889,E2 26530.889} C_VEL
LIN {X 0,Y 572.295,Z 1218.057,A -85,B 0,C 180,E1 26529.014,E2 26529.014} C_VEL
LIN {X 0,Y 573.862,Z 1201.125,A -85,B 0,C 180,E1 26527.083,E2 26527.083} C_VEL
LIN {X 0,Y 575.788,Z 1181.343,A -85,B 0,C 180,E1 26525.152,E2 26525.152} C_VEL
LIN {X 0,Y 577.691,Z 1162.07,A -85,B 0,C 180,E1 26523.534,E2 26523.534} C_VEL
LIN {X 0,Y 579.74,Z 1142.246,A -85,B 0,C 180,E1 26522.08,E2 26522.08} C_VEL
LIN {X 0,Y 581.871,Z 1120.779,A -85,B 0,C 180,E1 26520.735,E2 26520.735} C_VEL
LIN {X 0,Y 583.969,Z 1099.885,A -85,B 0,C 180,E1 26519.607,E2 26519.607} C_VEL
LIN {X 0,Y 586.093,Z 1077.421,A -85,B 0,C 180,E1 26518.59,E2 26518.59} C_VEL
LIN {X 0,Y 587.966,Z 1056.693,A -85,B 0,C 180,E1 26517.809,E2 26517.809} C_VEL
LIN {X 0,Y 590.083,Z 1031.024,A -85,B 0,C 180,E1 26517.037,E2 26517.037} C_VEL
LIN {X 0,Y 591.665,Z 1009.109,A -85,B 0,C 180,E1 26516.539,E2 26516.539} C_VEL
LIN {X 0,Y 593.066,Z 977.162,A -85,B 0,C 180,E1 26516.012,E2 26516.012} C_VEL
LIN {X 0,Y 594.806,Z 961.072,A -85,B 0,C 180,E1 26515.847,E2 26515.847} C_VEL
LIN {X 0,Y 595.287,Z 957.652,A -85,B 0,C 180,E1 26515.818,E2 26515.818} C_VEL
LIN {X 0,Y 602.097,Z 945.328,A -85,B 0,C 180,E1 26515.163,E2 26515.163} C_VEL
LIN {X 0,Y 613.532,Z 927.397,A -85,B 0,C 180,E1 26514.309,E2 26514.309} C_VEL
LIN {X 0,Y 623.103,Z 914.802,A -85,B 0,C 180,E1 26513.808,E2 26513.808} C_VEL
LIN {X 0,Y 612.93,Z 904.803,A -85,B 0,C 180,E1 26512.451,E2 26512.451} C_VEL
LIN {X 0,Y 604.861,Z 893.938,A -85,B 0,C 180,E1 26511.087,E2 26511.087} C_VEL
LIN {X 0,Y 598.336,Z 881.421,A -85,B 0,C 180,E1 26509.644,E2 26509.644} C_VEL
LIN {X 0,Y 593.552,Z 867.327,A -85,B 0,C 180,E1 26508.124,E2 26508.124} C_VEL
LIN {X 0,Y 590.761,Z 851.943,A -85,B 0,C 180,E1 26506.596,E2 26506.596} C_VEL
LIN {X 0,Y 589.95,Z 833.54,A -85,B 0,C 180,E1 26504.893,E2 26504.893} C_VEL
LIN {X 0,Y 593.876,Z 781.89,A -85,B 0,C 180,E1 26500.449,E2 26500.449} C_VEL
LIN {X 0,Y 596.93,Z 747.033,A -85,B 0,C 180,E1 26497.394,E2 26497.394} C_VEL
LIN {X 0,Y 599.927,Z 713.189,A -85,B 0,C 180,E1 26494.345,E2 26494.345} C_VEL
LIN {X 0,Y 601.818,Z 691.035,A -85,B 0,C 180,E1 26492.287,E2 26492.287} C_VEL
LIN {X 0,Y 593.529,Z 671.123,A -85,B 0,C 180,E1 26489.356,E2 26489.356} C_VEL
LIN {X 0,Y 585.857,Z 653.392,A -85,B 0,C 180,E1 26486.562,E2 26486.562} C_VEL
LIN {X 0,Y 578.309,Z 636.847,A -85,B 0,C 180,E1 26483.757,E2 26483.757} C_VEL
LIN {X 0,Y 573.075,Z 625.37,A -85,B 0,C 180,E1 26481.709,E2 26481.709} C_VEL
LIN {X 0,Y 570.779,Z 620.68,A -85,B 0,C 180,E1 26480.831,E2 26480.831} C_VEL
LIN {X 0,Y 569.385,Z 617.055,A -85,B 0,C 180,E1 26480.186,E2 26480.186} C_VEL
LIN {X 0,Y 569.367,Z 617.053,A -85,B 0,C 180,E1 26476.844,E2 26476.844} C_VEL
LIN {X 0,Y 569.376,Z 617.057,A -85,B 0,C 180,E1 26473.611,E2 26473.611} C_VEL
LIN {X 0,Y 569.367,Z 617.053,A -85,B 0,C 180,E1 26470.319,E2 26470.319} C_VEL
LIN {X 0,Y 569.381,Z 617.056,A -85,B 0,C 180,E1 26466.96,E2 26466.96} C_VEL
LIN {X 0,Y 569.374,Z 617.052,A -85,B 0,C 180,E1 26463.625,E2 26463.625} C_VEL
LIN {X 0,Y 569.376,Z 617.057,A -85,B 0,C 180,E1 26460.302,E2 26460.302} C_VEL
LIN {X 0,Y 569.365,Z 617.059,A -85,B 0,C 180,E1 26456.98,E2 26456.98} C_VEL
LIN {X 0,Y 569.371,Z 617.056,A -85,B 0,C 180,E1 26453.685,E2 26453.685} C_VEL
LIN {X 0,Y 569.368,Z 617.054,A -85,B 0,C 180,E1 26450.396,E2 26450.396} C_VEL
LIN {X 0,Y 569.382,Z 617.051,A -85,B 0,C 180,E1 26447.01,E2 26447.01} C_VEL
LIN {X 0,Y 569.373,Z 617.053,A -85,B 0,C 180,E1 26443.681,E2 26443.681} C_VEL
LIN {X 0,Y 569.374,Z 617.055,A -85,B 0,C 180,E1 26440.402,E2 26440.402} C_VEL
LIN {X 0,Y 569.366,Z 617.057,A -85,B 0,C 180,E1 26437.163,E2 26437.163} C_VEL
LIN {X 0,Y 569.369,Z 617.058,A -85,B 0,C 180,E1 26433.958,E2 26433.958} C_VEL
LIN {X 0,Y 569.367,Z 617.058,A -85,B 0,C 180,E1 26430.777,E2 26430.777} C_VEL
LIN {X 0,Y 569.374,Z 617.056,A -85,B 0,C 180,E1 26427.448,E2 26427.448} C_VEL
LIN {X 0,Y 569.38,Z 617.052,A -85,B 0,C 180,E1 26424.088,E2 26424.088} C_VEL
LIN {X 0,Y 569.385,Z 617.051,A -85,B 0,C 180,E1 26420.751,E2 26420.751} C_VEL
LIN {X 0,Y 569.37,Z 617.035,A -85,B 0,C 180,E1 26417.459,E2 26417.459} C_VEL
LIN {X 0,Y 569.382,Z 617.059,A -85,B 0,C 180,E1 26414.198,E2 26414.198} C_VEL
LIN {X 0,Y 569.373,Z 617.044,A -85,B 0,C 180,E1 26410.787,E2 26410.787} C_VEL
LIN {X 0,Y 569.38,Z 617.042,A -85,B 0,C 180,E1 26407.415,E2 26407.415} C_VEL
LIN {X 0,Y 569.405,Z 617.209,A -85,B 0,C 180,E1 26405.084,E2 26405.084} C_VEL
LIN {X 0,Y 578.235,Z 643.458,A -85,B 0,C 180,E1 26402.735,E2 26402.735} C_VEL
LIN {X 0,Y 581.481,Z 654.898,A -85,B 0,C 180,E1 26401.746,E2 26401.746} C_VEL
LIN {X 0,Y 580.129,Z 698.725,A -85,B 0,C 180,E1 26398.628,E2 26398.628} C_VEL
LIN {X 0,Y 578.367,Z 746.016,A -85,B 0,C 180,E1 26395.222,E2 26395.222} C_VEL
LIN {X 0,Y 577.684,Z 764.311,A -85,B 0,C 180,E1 26393.909,E2 26393.909} C_VEL
LIN {X 0,Y 576.526,Z 770.763,A -85,B 0,C 180,E1 26393.496,E2 26393.496} C_VEL
LIN {X 0,Y 570.118,Z 788.502,A -85,B 0,C 180,E1 26392.514,E2 26392.514} C_VEL
LIN {X 0,Y 569.252,Z 794.06,A -85,B 0,C 180,E1 26392.154,E2 26392.154} C_VEL
LIN {X 0,Y 568.085,Z 837.887,A -85,B 0,C 180,E1 26389.154,E2 26389.154} C_VEL
LIN {X 0,Y 568.054,Z 844.137,A -85,B 0,C 180,E1 26388.764,E2 26388.764} C_VEL
LIN {X 0,Y 568.804,Z 852.24,A -85,B 0,C 180,E1 26388.63,E2 26388.63} C_VEL
LIN {X 0,Y 567.123,Z 1013.737,A -85,B 0,C 180,E1 26386.542,E2 26386.542} C_VEL
LIN {X 0,Y 566.883,Z 1031.229,A -85,B 0,C 180,E1 26386.131,E2 26386.131} C_VEL
LIN {X 0,Y 566.439,Z 1047.443,A -85,B 0,C 180,E1 26385.562,E2 26385.562} C_VEL
LIN {X 0,Y 565.813,Z 1063.752,A -85,B 0,C 180,E1 26384.793,E2 26384.793} C_VEL
LIN {X 0,Y 565.081,Z 1078.98,A -85,B 0,C 180,E1 26383.871,E2 26383.871} C_VEL
LIN {X 0,Y 564.289,Z 1093.123,A -85,B 0,C 180,E1 26382.795,E2 26382.795} C_VEL
LIN {X 0,Y 563.477,Z 1106.162,A -85,B 0,C 180,E1 26381.566,E2 26381.566} C_VEL
LIN {X 0,Y 562.727,Z 1117.699,A -85,B 0,C 180,E1 26380.233,E2 26380.233} C_VEL
LIN {X 0,Y 562.074,Z 1127.818,A -85,B 0,C 180,E1 26378.799,E2 26378.799} C_VEL
LIN {X 0,Y 561.533,Z 1136.497,A -85,B 0,C 180,E1 26377.262,E2 26377.262} C_VEL
LIN {X 0,Y 561.121,Z 1143.718,A -85,B 0,C 180,E1 26375.623,E2 26375.623} C_VEL
LIN {X 0,Y 560.837,Z 1149.437,A -85,B 0,C 180,E1 26373.883,E2 26373.883} C_VEL
LIN {X 0,Y 560.67,Z 1153.347,A -85,B 0,C 180,E1 26372.145,E2 26372.145} C_VEL
LIN {X 0,Y 560.588,Z 1155.592,A -85,B 0,C 180,E1 26370.305,E2 26370.305} C_VEL
LIN {X 0,Y 560.569,Z 1156.035,A -85,B 0,C 180,E1 26368.465,E2 26368.465} C_VEL
LIN {X 0,Y 560.627,Z 1154.701,A -85,B 0,C 180,E1 26366.625,E2 26366.625} C_VEL
LIN {X 0,Y 560.757,Z 1151.702,A -85,B 0,C 180,E1 26364.884,E2 26364.884} C_VEL
LIN {X 0,Y 560.998,Z 1146.814,A -85,B 0,C 180,E1 26363.106,E2 26363.106} C_VEL
LIN {X 0,Y 561.36,Z 1140.257,A -85,B 0,C 180,E1 26361.394,E2 26361.394} C_VEL
LIN {X 0,Y 561.864,Z 1132.138,A -85,B 0,C 180,E1 26359.776,E2 26359.776} C_VEL
LIN {X 0,Y 562.474,Z 1122.79,A -85,B 0,C 180,E1 26358.307,E2 26358.307} C_VEL
LIN {X 0,Y 563.239,Z 1111.441,A -85,B 0,C 180,E1 26356.865,E2 26356.865} C_VEL
LIN {X 0,Y 564.058,Z 1098.97,A -85,B 0,C 180,E1 26355.577,E2 26355.577} C_VEL
LIN {X 0,Y 564.876,Z 1085.414,A -85,B 0,C 180,E1 26354.443,E2 26354.443} C_VEL
LIN {X 0,Y 565.637,Z 1070.87,A -85,B 0,C 180,E1 26353.464,E2 26353.464} C_VEL
LIN {X 0,Y 566.319,Z 1055.396,A -85,B 0,C 180,E1 26352.638,E2 26352.638} C_VEL
LIN {X 0,Y 566.881,Z 1038.751,A -85,B 0,C 180,E1 26351.961,E2 26351.961} C_VEL
LIN {X 0,Y 567.23,Z 1021.463,A -85,B 0,C 180,E1 26351.469,E2 26351.469} C_VEL
LIN {X 0,Y 567.372,Z 1002.009,A -85,B 0,C 180,E1 26351.134,E2 26351.134} C_VEL
LIN {X 0,Y 568.847,Z 848.414,A -85,B 0,C 180,E1 26349.16,E2 26349.16} C_VEL
LIN {X 0,Y 568.188,Z 843.606,A -85,B 0,C 180,E1 26349.068,E2 26349.068} C_VEL
LIN {X 0,Y 569.413,Z 797.377,A -85,B 0,C 180,E1 26345.908,E2 26345.908} C_VEL
LIN {X 0,Y 571.1,Z 751.753,A -85,B 0,C 180,E1 26342.638,E2 26342.638} C_VEL
LIN {X 0,Y 572.897,Z 706.584,A -85,B 0,C 180,E1 26339.359,E2 26339.359} C_VEL
LIN {X 0,Y 574.392,Z 665.379,A -85,B 0,C 180,E1 26336.387,E2 26336.387} C_VEL
LIN {X 0,Y 574.424,Z 656.903,A -85,B 0,C 180,E1 26335.774,E2 26335.774} C_VEL
LIN {X 0,Y 567.309,Z 634.567,A -85,B 0,C 180,E1 26333.741,E2 26333.741} C_VEL
LIN {X 0,Y 561.432,Z 618.045,A -85,B 0,C 180,E1 26332.185,E2 26332.185} C_VEL
LIN {X 0,Y 561.438,Z 618.033,A -85,B 0,C 180,E1 26328.881,E2 26328.881} C_VEL
LIN {X 0,Y 561.431,Z 618.049,A -85,B 0,C 180,E1 26325.575,E2 26325.575} C_VEL
LIN {X 0,Y 561.442,Z 618.042,A -85,B 0,C 180,E1 26322.176,E2 26322.176} C_VEL
LIN {X 0,Y 561.456,Z 618.086,A -85,B 0,C 180,E1 26319.148,E2 26319.148} C_VEL
LIN {X 0,Y 562.515,Z 621.182,A -85,B 0,C 180,E1 26318.707,E2 26318.707} C_VEL
LIN {X 0,Y 566.94,Z 630.603,A -85,B 0,C 180,E1 26317.305,E2 26317.305} C_VEL
LIN {X 0,Y 588.306,Z 661.91,A -85,B 0,C 180,E1 26314.993,E2 26314.993} C_VEL
LIN {X 0,Y 591.933,Z 667.788,A -85,B 0,C 180,E1 26314.617,E2 26314.617} C_VEL
LIN {X 0,Y 584.154,Z 906.028,A -85,B 0,C 180,E1 26311.053,E2 26311.053} C_VEL
LIN {X 0,Y 582.583,Z 962.421,A -85,B 0,C 180,E1 26310.198,E2 26310.198} C_VEL
LIN {X 0,Y 581.546,Z 985.501,A -85,B 0,C 180,E1 26309.66,E2 26309.66} C_VEL
LIN {X 0,Y 580.188,Z 1008.678,A -85,B 0,C 180,E1 26308.937,E2 26308.937} C_VEL
LIN {X 0,Y 578.644,Z 1030.12,A -85,B 0,C 180,E1 26308.091,E2 26308.091} C_VEL
LIN {X 0,Y 576.755,Z 1051.456,A -85,B 0,C 180,E1 26307.052,E2 26307.052} C_VEL
LIN {X 0,Y 574.676,Z 1073.099,A -85,B 0,C 180,E1 26305.784,E2 26305.784} C_VEL
LIN {X 0,Y 572.705,Z 1091.708,A -85,B 0,C 180,E1 26304.498,E2 26304.498} C_VEL
LIN {X 0,Y 570.598,Z 1110.156,A -85,B 0,C 180,E1 26303.003,E2 26303.003} C_VEL
LIN {X 0,Y 568.583,Z 1127.807,A -85,B 0,C 180,E1 26301.348,E2 26301.348} C_VEL
LIN {X 0,Y 566.783,Z 1143.009,A -85,B 0,C 180,E1 26299.691,E2 26299.691} C_VEL
LIN {X 0,Y 565.013,Z 1158.661,A -85,B 0,C 180,E1 26297.721,E2 26297.721} C_VEL
LIN {X 0,Y 563.57,Z 1172.146,A -85,B 0,C 180,E1 26295.751,E2 26295.751} C_VEL
LIN {X 0,Y 562.372,Z 1184.166,A -85,B 0,C 180,E1 26293.679,E2 26293.679} C_VEL
LIN {X 0,Y 561.443,Z 1194.95,A -85,B 0,C 180,E1 26291.506,E2 26291.506} C_VEL
LIN {X 0,Y 560.796,Z 1203.843,A -85,B 0,C 180,E1 26289.338,E2 26289.338} C_VEL
LIN {X 0,Y 560.357,Z 1211.765,A -85,B 0,C 180,E1 26286.969,E2 26286.969} C_VEL
LIN {X 0,Y 560.119,Z 1217.661,A -85,B 0,C 180,E1 26284.71,E2 26284.71} C_VEL
LIN {X 0,Y 560,Z 1222.113,A -85,B 0,C 180,E1 26282.354,E2 26282.354} C_VEL
LIN {X 0,Y 559.974,Z 1224.908,A -85,B 0,C 180,E1 26280.102,E2 26280.102} C_VEL
LIN {X 0,Y 559.948,Z 1226.179,A -85,B 0,C 180,E1 26277.851,E2 26277.851} C_VEL
LIN {X 0,Y 559.947,Z 1226.092,A -85,B 0,C 180,E1 26275.596,E2 26275.596} C_VEL
LIN {X 0,Y 559.968,Z 1224.382,A -85,B 0,C 180,E1 26273.232,E2 26273.232} C_VEL
LIN {X 0,Y 560.035,Z 1221.093,A -85,B 0,C 180,E1 26270.857,E2 26270.857} C_VEL
LIN {X 0,Y 560.168,Z 1216.563,A -85,B 0,C 180,E1 26268.676,E2 26268.676} C_VEL
LIN {X 0,Y 560.471,Z 1209.902,A -85,B 0,C 180,E1 26266.274,E2 26266.274} C_VEL
LIN {X 0,Y 560.919,Z 1202.547,A -85,B 0,C 180,E1 26264.173,E2 26264.173} C_VEL
LIN {X 0,Y 561.638,Z 1192.998,A -85,B 0,C 180,E1 26261.954,E2 26261.954} C_VEL
LIN {X 0,Y 562.604,Z 1182.127,A -85,B 0,C 180,E1 26259.831,E2 26259.831} C_VEL
LIN {X 0,Y 563.708,Z 1170.411,A -85,B 0,C 180,E1 26257.911,E2 26257.911} C_VEL
LIN {X 0,Y 565.205,Z 1155.967,A -85,B 0,C 180,E1 26255.879,E2 26255.879} C_VEL
LIN {X 0,Y 566.752,Z 1141.459,A -85,B 0,C 180,E1 26254.129,E2 26254.129} C_VEL
LIN {X 0,Y 568.407,Z 1125.69,A -85,B 0,C 180,E1 26252.499,E2 26252.499} C_VEL
LIN {X 0,Y 570.145,Z 1108.61,A -85,B 0,C 180,E1 26250.967,E2 26250.967} C_VEL
LIN {X 0,Y 571.778,Z 1091.2,A -85,B 0,C 180,E1 26249.643,E2 26249.643} C_VEL
LIN {X 0,Y 573.493,Z 1071.161,A -85,B 0,C 180,E1 26248.345,E2 26248.345} C_VEL
LIN {X 0,Y 574.964,Z 1051.117,A -85,B 0,C 180,E1 26247.259,E2 26247.259} C_VEL
LIN {X 0,Y 576.123,Z 1031.085,A -85,B 0,C 180,E1 26246.383,E2 26246.383} C_VEL
LIN {X 0,Y 577.117,Z 1009.182,A -85,B 0,C 180,E1 26245.614,E2 26245.614} C_VEL
LIN {X 0,Y 577.704,Z 988.926,A -85,B 0,C 180,E1 26245.074,E2 26245.074} C_VEL
LIN {X 0,Y 577.993,Z 966.73,A -85,B 0,C 180,E1 26244.662,E2 26244.662} C_VEL
LIN {X 0,Y 579.655,Z 829.969,A -85,B 0,C 180,E1 26242.933,E2 26242.933} C_VEL
LIN {X 0,Y 581.892,Z 729.55,A -85,B 0,C 180,E1 26241.493,E2 26241.493} C_VEL
LIN {X 0,Y 582.936,Z 692.589,A -85,B 0,C 180,E1 26240.911,E2 26240.911} C_VEL
LIN {X 0,Y 579.822,Z 692.27,A -85,B 0,C 180,E1 26240.664,E2 26240.664} C_VEL
LIN {X 0,Y 579.291,Z 692.13,A -85,B 0,C 180,E1 26240.607,E2 26240.607} C_VEL
LIN {X 0,Y 574.165,Z 703.576,A -85,B 0,C 180,E1 26239.172,E2 26239.172} C_VEL
LIN {X 0,Y 570.205,Z 716.931,A -85,B 0,C 180,E1 26237.733,E2 26237.733} C_VEL
LIN {X 0,Y 566.919,Z 734.106,A -85,B 0,C 180,E1 26236.12,E2 26236.12} C_VEL
LIN {X 0,Y 564.366,Z 756.302,A -85,B 0,C 180,E1 26234.293,E2 26234.293} C_VEL
LIN {X 0,Y 563.134,Z 782.4,A -85,B 0,C 180,E1 26232.34,E2 26232.34} C_VEL
LIN {X 0,Y 564.126,Z 803.528,A -85,B 0,C 180,E1 26230.813,E2 26230.813} C_VEL
LIN {X 0,Y 567.194,Z 823.438,A -85,B 0,C 180,E1 26229.394,E2 26229.394} C_VEL
LIN {X 0,Y 572.09,Z 841.159,A -85,B 0,C 180,E1 26228.14,E2 26228.14} C_VEL
LIN {X 0,Y 579.184,Z 858.474,A -85,B 0,C 180,E1 26226.927,E2 26226.927} C_VEL
LIN {X 0,Y 587.813,Z 874.144,A -85,B 0,C 180,E1 26225.851,E2 26225.851} C_VEL
LIN {X 0,Y 598.305,Z 888.953,A -85,B 0,C 180,E1 26224.859,E2 26224.859} C_VEL
LIN {X 0,Y 606.824,Z 899.074,A -85,B 0,C 180,E1 26224.201,E2 26224.201} C_VEL
LIN {X 0,Y 596.911,Z 912.041,A -85,B 0,C 180,E1 26223.502,E2 26223.502} C_VEL
LIN {X 0,Y 590.987,Z 921.644,A -85,B 0,C 180,E1 26222.986,E2 26222.986} C_VEL
LIN {X 0,Y 584.786,Z 939.044,A -85,B 0,C 180,E1 26223.016,E2 26223.016} C_VEL
LIN {X 0,Y 579.806,Z 958.068,A -85,B 0,C 180,E1 26222.971,E2 26222.971} C_VEL
LIN {X 0,Y 577.695,Z 972.284,A -85,B 0,C 180,E1 26222.819,E2 26222.819} C_VEL
LIN {X 0,Y 576.264,Z 1003.162,A -85,B 0,C 180,E1 26222.203,E2 26222.203} C_VEL
LIN {X 0,Y 574.594,Z 1033.749,A -85,B 0,C 180,E1 26221.398,E2 26221.398} C_VEL
LIN {X 0,Y 573.025,Z 1062.823,A -85,B 0,C 180,E1 26220.435,E2 26220.435} C_VEL
LIN {X 0,Y 571.539,Z 1090.194,A -85,B 0,C 180,E1 26219.332,E2 26219.332} C_VEL
LIN {X 0,Y 570.141,Z 1114.85,A -85,B 0,C 180,E1 26218.15,E2 26218.15} C_VEL
LIN {X 0,Y 568.742,Z 1138.72,A -85,B 0,C 180,E1 26216.805,E2 26216.805} C_VEL
LIN {X 0,Y 567.314,Z 1161.736,A -85,B 0,C 180,E1 26215.289,E2 26215.289} C_VEL
LIN {X 0,Y 565.995,Z 1181.668,A -85,B 0,C 180,E1 26213.754,E2 26213.754} C_VEL
LIN {X 0,Y 564.737,Z 1200.711,A -85,B 0,C 180,E1 26212.047,E2 26212.047} C_VEL
LIN {X 0,Y 563.637,Z 1216.985,A -85,B 0,C 180,E1 26210.348,E2 26210.348} C_VEL
LIN {X 0,Y 562.607,Z 1232.587,A -85,B 0,C 180,E1 26208.443,E2 26208.443} C_VEL
LIN {X 0,Y 561.779,Z 1245.795,A -85,B 0,C 180,E1 26206.547,E2 26206.547} C_VEL
LIN {X 0,Y 561.121,Z 1257.446,A -85,B 0,C 180,E1 26204.553,E2 26204.553} C_VEL
LIN {X 0,Y 560.649,Z 1266.691,A -85,B 0,C 180,E1 26202.673,E2 26202.673} C_VEL
LIN {X 0,Y 560.338,Z 1274.377,A -85,B 0,C 180,E1 26200.8,E2 26200.8} C_VEL
LIN {X 0,Y 560.103,Z 1282.143,A -85,B 0,C 180,E1 26198.419,E2 26198.419} C_VEL
LIN {X 0,Y 559.998,Z 1287.291,A -85,B 0,C 180,E1 26196.254,E2 26196.254} C_VEL
LIN {X 0,Y 559.95,Z 1290.625,A -85,B 0,C 180,E1 26194.302,E2 26194.302} C_VEL
LIN {X 0,Y 559.938,Z 1292.81,A -85,B 0,C 180,E1 26192.253,E2 26192.253} C_VEL
LIN {X 0,Y 559.942,Z 1293.711,A -85,B 0,C 180,E1 26189.899,E2 26189.899} C_VEL
LIN {X 0,Y 559.926,Z 1292.782,A -85,B 0,C 180,E1 26187.545,E2 26187.545} C_VEL
LIN {X 0,Y 559.934,Z 1290.595,A -85,B 0,C 180,E1 26185.495,E2 26185.495} C_VEL
LIN {X 0,Y 559.977,Z 1287.095,A -85,B 0,C 180,E1 26183.44,E2 26183.44} C_VEL
LIN {X 0,Y 560.097,Z 1281.683,A -85,B 0,C 180,E1 26181.17,E2 26181.17} C_VEL
LIN {X 0,Y 560.348,Z 1274.436,A -85,B 0,C 180,E1 26178.89,E2 26178.89} C_VEL
LIN {X 0,Y 560.737,Z 1266.203,A -85,B 0,C 180,E1 26176.808,E2 26176.808} C_VEL
LIN {X 0,Y 561.332,Z 1256.322,A -85,B 0,C 180,E1 26174.716,E2 26174.716} C_VEL
LIN {X 0,Y 562.218,Z 1243.935,A -85,B 0,C 180,E1 26172.51,E2 26172.51} C_VEL
LIN {X 0,Y 563.367,Z 1229.955,A -85,B 0,C 180,E1 26170.402,E2 26170.402} C_VEL
LIN {X 0,Y 564.819,Z 1214.072,A -85,B 0,C 180,E1 26168.342,E2 26168.342} C_VEL
LIN {X 0,Y 566.708,Z 1194.983,A -85,B 0,C 180,E1 26166.226,E2 26166.226} C_VEL
LIN {X 0,Y 568.768,Z 1174.88,A -85,B 0,C 180,E1 26164.322,E2 26164.322} C_VEL
LIN {X 0,Y 571.058,Z 1153.453,A -85,B 0,C 180,E1 26162.583,E2 26162.583} C_VEL
LIN {X 0,Y 573.214,Z 1132.967,A -85,B 0,C 180,E1 26161.165,E2 26161.165} C_VEL
LIN {X 0,Y 575.545,Z 1111.376,A -85,B 0,C 180,E1 26159.865,E2 26159.865} C_VEL
LIN {X 0,Y 577.817,Z 1088.813,A -85,B 0,C 180,E1 26158.728,E2 26158.728} C_VEL
LIN {X 0,Y 580.104,Z 1066.134,A -85,B 0,C 180,E1 26157.762,E2 26157.762} C_VEL
LIN {X 0,Y 582.234,Z 1042.654,A -85,B 0,C 180,E1 26156.966,E2 26156.966} C_VEL
LIN {X 0,Y 584.21,Z 1019.135,A -85,B 0,C 180,E1 26156.331,E2 26156.331} C_VEL
LIN {X 0,Y 585.719,Z 994.471,A -85,B 0,C 180,E1 26155.849,E2 26155.849} C_VEL
LIN {X 0,Y 586.962,Z 970.732,A -85,B 0,C 180,E1 26155.494,E2 26155.494} C_VEL
LIN {X 0,Y 589.075,Z 955.78,A -85,B 0,C 180,E1 26155.348,E2 26155.348} C_VEL
LIN {X 0,Y 596.426,Z 942.818,A -85,B 0,C 180,E1 26154.665,E2 26154.665} C_VEL
LIN {X 0,Y 607.538,Z 925.537,A -85,B 0,C 180,E1 26153.844,E2 26153.844} C_VEL
LIN {X 0,Y 613.76,Z 917.026,A -85,B 0,C 180,E1 26153.488,E2 26153.488} C_VEL
LIN {X 0,Y 604.222,Z 906.843,A -85,B 0,C 180,E1 26152.126,E2 26152.126} C_VEL
LIN {X 0,Y 596.577,Z 895.655,A -85,B 0,C 180,E1 26150.745,E2 26150.745} C_VEL
LIN {X 0,Y 590.237,Z 882.408,A -85,B 0,C 180,E1 26149.222,E2 26149.222} C_VEL
LIN {X 0,Y 585.775,Z 867.728,A -85,B 0,C 180,E1 26147.656,E2 26147.656} C_VEL
LIN {X 0,Y 583.361,Z 851.489,A -85,B 0,C 180,E1 26146.045,E2 26146.045} C_VEL
LIN {X 0,Y 583.001,Z 832.144,A -85,B 0,C 180,E1 26144.27,E2 26144.27} C_VEL
LIN {X 0,Y 586.815,Z 786.566,A -85,B 0,C 180,E1 26140.325,E2 26140.325} C_VEL
LIN {X 0,Y 590.11,Z 750.877,A -85,B 0,C 180,E1 26137.167,E2 26137.167} C_VEL
LIN {X 0,Y 593.257,Z 716.875,A -85,B 0,C 180,E1 26134.084,E2 26134.084} C_VEL
LIN {X 0,Y 595.26,Z 695.114,A -85,B 0,C 180,E1 26132.06,E2 26132.06} C_VEL
LIN {X 0,Y 587.407,Z 676.149,A -85,B 0,C 180,E1 26129.244,E2 26129.244} C_VEL
LIN {X 0,Y 579.753,Z 658.374,A -85,B 0,C 180,E1 26126.421,E2 26126.421} C_VEL
LIN {X 0,Y 572.499,Z 642.317,A -85,B 0,C 180,E1 26123.685,E2 26123.685} C_VEL
LIN {X 0,Y 566.948,Z 630.337,A -85,B 0,C 180,E1 26121.521,E2 26121.521} C_VEL
LIN {X 0,Y 563.052,Z 621.951,A -85,B 0,C 180,E1 26119.936,E2 26119.936} C_VEL
LIN {X 0,Y 561.567,Z 618.765,A -85,B 0,C 180,E1 26119.327,E2 26119.327} C_VEL
LIN {X 0,Y 561.439,Z 618.041,A -85,B 0,C 180,E1 26119.188,E2 26119.188} C_VEL
LIN {X 0,Y 561.43,Z 618.048,A -85,B 0,C 180,E1 26115.812,E2 26115.812} C_VEL
LIN {X 0,Y 561.426,Z 618.043,A -85,B 0,C 180,E1 26112.549,E2 26112.549} C_VEL
LIN {X 0,Y 561.428,Z 618.046,A -85,B 0,C 180,E1 26109.224,E2 26109.224} C_VEL
LIN {X 0,Y 561.433,Z 618.038,A -85,B 0,C 180,E1 26105.929,E2 26105.929} C_VEL
LIN {X 0,Y 561.437,Z 618.046,A -85,B 0,C 180,E1 26102.45,E2 26102.45} C_VEL
LIN {X 0,Y 561.446,Z 618.043,A -85,B 0,C 180,E1 26099.082,E2 26099.082} C_VEL
LIN {X 0,Y 561.439,Z 618.04,A -85,B 0,C 180,E1 26095.71,E2 26095.71} C_VEL
LIN {X 0,Y 561.442,Z 618.041,A -85,B 0,C 180,E1 26092.324,E2 26092.324} C_VEL
LIN {X 0,Y 561.435,Z 618.046,A -85,B 0,C 180,E1 26088.892,E2 26088.892} C_VEL
LIN {X 0,Y 561.427,Z 618.046,A -85,B 0,C 180,E1 26085.562,E2 26085.562} C_VEL
LIN {X 0,Y 561.427,Z 618.046,A -85,B 0,C 180,E1 26082.269,E2 26082.269} C_VEL
LIN {X 0,Y 561.433,Z 618.044,A -85,B 0,C 180,E1 26078.937,E2 26078.937} C_VEL
LIN {X 0,Y 561.441,Z 618.041,A -85,B 0,C 180,E1 26075.508,E2 26075.508} C_VEL
LIN {X 0,Y 561.451,Z 618.038,A -85,B 0,C 180,E1 26072.042,E2 26072.042} C_VEL
LIN {X 0,Y 561.445,Z 618.038,A -85,B 0,C 180,E1 26068.666,E2 26068.666} C_VEL
LIN {X 0,Y 561.44,Z 618.036,A -85,B 0,C 180,E1 26065.257,E2 26065.257} C_VEL
LIN {X 0,Y 561.435,Z 618.039,A -85,B 0,C 180,E1 26061.83,E2 26061.83} C_VEL
LIN {X 0,Y 561.428,Z 618.042,A -85,B 0,C 180,E1 26058.507,E2 26058.507} C_VEL
LIN {X 0,Y 561.43,Z 618.037,A -85,B 0,C 180,E1 26055.137,E2 26055.137} C_VEL
LIN {X 0,Y 561.43,Z 618.026,A -85,B 0,C 180,E1 26051.888,E2 26051.888} C_VEL
LIN {X 0,Y 561.441,Z 618.042,A -85,B 0,C 180,E1 26048.557,E2 26048.557} C_VEL
LIN {X 0,Y 561.469,Z 618.269,A -85,B 0,C 180,E1 26045.487,E2 26045.487} C_VEL
LIN {X 0,Y 570.195,Z 643.785,A -85,B 0,C 180,E1 26043.168,E2 26043.168} C_VEL
LIN {X 0,Y 574.161,Z 657.471,A -85,B 0,C 180,E1 26041.963,E2 26041.963} C_VEL
LIN {X 0,Y 572.79,Z 699.102,A -85,B 0,C 180,E1 26038.978,E2 26038.978} C_VEL
LIN {X 0,Y 570.986,Z 746.184,A -85,B 0,C 180,E1 26035.571,E2 26035.571} C_VEL
LIN {X 0,Y 569.265,Z 793.616,A -85,B 0,C 180,E1 26032.186,E2 26032.186} C_VEL
LIN {X 0,Y 569.252,Z 794.06,A -85,B 0,C 180,E1 26032.154,E2 26032.154} C_VEL
LIN {X 0,Y 568.139,Z 800.567,A -85,B 0,C 180,E1 26031.743,E2 26031.743} C_VEL
LIN {X 0,Y 561.775,Z 818.475,A -85,B 0,C 180,E1 26030.773,E2 26030.773} C_VEL
LIN {X 0,Y 560.915,Z 824.096,A -85,B 0,C 180,E1 26030.417,E2 26030.417} C_VEL
LIN {X 0,Y 560.531,Z 844.972,A -85,B 0,C 180,E1 26029.036,E2 26029.036} C_VEL
LIN {X 0,Y 561.283,Z 853.007,A -85,B 0,C 180,E1 26028.9,E2 26028.9} C_VEL
LIN {X 0,Y 559.516,Z 1014.609,A -85,B 0,C 180,E1 26026.783,E2 26026.783} C_VEL
LIN {X 0,Y 559.269,Z 1032.14,A -85,B 0,C 180,E1 26026.367,E2 26026.367} C_VEL
LIN {X 0,Y 558.801,Z 1048.597,A -85,B 0,C 180,E1 26025.781,E2 26025.781} C_VEL
LIN {X 0,Y 558.151,Z 1064.865,A -85,B 0,C 180,E1 26025.001,E2 26025.001} C_VEL
LIN {X 0,Y 557.387,Z 1080.065,A -85,B 0,C 180,E1 26024.066,E2 26024.066} C_VEL
LIN {X 0,Y 556.559,Z 1094.176,A -85,B 0,C 180,E1 26022.976,E2 26022.976} C_VEL
LIN {X 0,Y 555.708,Z 1107.199,A -85,B 0,C 180,E1 26021.73,E2 26021.73} C_VEL
LIN {X 0,Y 554.878,Z 1119.374,A -85,B 0,C 180,E1 26020.296,E2 26020.296} C_VEL
LIN {X 0,Y 554.187,Z 1129.477,A -85,B 0,C 180,E1 26018.82,E2 26018.82} C_VEL
LIN {X 0,Y 553.588,Z 1138.484,A -85,B 0,C 180,E1 26017.158,E2 26017.158} C_VEL
LIN {X 0,Y 553.158,Z 1145.873,A -85,B 0,C 180,E1 26015.392,E2 26015.392} C_VEL
LIN {X 0,Y 552.879,Z 1151.246,A -85,B 0,C 180,E1 26013.628,E2 26013.628} C_VEL
LIN {X 0,Y 552.708,Z 1154.792,A -85,B 0,C 180,E1 26011.865,E2 26011.865} C_VEL
LIN {X 0,Y 552.642,Z 1156.747,A -85,B 0,C 180,E1 26009.999,E2 26009.999} C_VEL
LIN {X 0,Y 552.634,Z 1156.918,A -85,B 0,C 180,E1 26008.132,E2 26008.132} C_VEL
LIN {X 0,Y 552.706,Z 1155.211,A -85,B 0,C 180,E1 26006.265,E2 26006.265} C_VEL
LIN {X 0,Y 552.879,Z 1151.658,A -85,B 0,C 180,E1 26004.394,E2 26004.394} C_VEL
LIN {X 0,Y 553.17,Z 1146.49,A -85,B 0,C 180,E1 26002.625,E2 26002.625} C_VEL
LIN {X 0,Y 553.573,Z 1139.768,A -85,B 0,C 180,E1 26000.958,E2 26000.958} C_VEL
LIN {X 0,Y 554.157,Z 1131.031,A -85,B 0,C 180,E1 25999.288,E2 25999.288} C_VEL
LIN {X 0,Y 554.837,Z 1121.441,A -85,B 0,C 180,E1 25997.827,E2 25997.827} C_VEL
LIN {X 0,Y 555.623,Z 1110.514,A -85,B 0,C 180,E1 25996.469,E2 25996.469} C_VEL
LIN {X 0,Y 556.492,Z 1097.539,A -85,B 0,C 180,E1 25995.166,E2 25995.166} C_VEL
LIN {X 0,Y 557.372,Z 1083.39,A -85,B 0,C 180,E1 25994.015,E2 25994.015} C_VEL
LIN {X 0,Y 558.197,Z 1068.181,A -85,B 0,C 180,E1 25993.022,E2 25993.022} C_VEL
LIN {X 0,Y 558.86,Z 1052.73,A -85,B 0,C 180,E1 25992.238,E2 25992.238} C_VEL
LIN {X 0,Y 559.39,Z 1035.683,A -85,B 0,C 180,E1 25991.588,E2 25991.588} C_VEL
LIN {X 0,Y 559.707,Z 1018.183,A -85,B 0,C 180,E1 25991.127,E2 25991.127} C_VEL
LIN {X 0,Y 559.87,Z 994.63,A -85,B 0,C 180,E1 25990.772,E2 25990.772} C_VEL
LIN {X 0,Y 561.37,Z 849.322,A -85,B 0,C 180,E1 25988.881,E2 25988.881} C_VEL
LIN {X 0,Y 560.712,Z 844.345,A -85,B 0,C 180,E1 25988.776,E2 25988.776} C_VEL
LIN {X 0,Y 561.984,Z 798.393,A -85,B 0,C 180,E1 25985.619,E2 25985.619} C_VEL
LIN {X 0,Y 563.74,Z 752.391,A -85,B 0,C 180,E1 25982.308,E2 25982.308} C_VEL
LIN {X 0,Y 565.637,Z 706.893,A -85,B 0,C 180,E1 25978.982,E2 25978.982} C_VEL
LIN {X 0,Y 567.169,Z 666.079,A -85,B 0,C 180,E1 25976.022,E2 25976.022} C_VEL
LIN {X 0,Y 567.282,Z 659.987,A -85,B 0,C 180,E1 25975.578,E2 25975.578} C_VEL
LIN {X 0,Y 560.169,Z 637.692,A -85,B 0,C 180,E1 25973.529,E2 25973.529} C_VEL
LIN {X 0,Y 553.496,Z 619.038,A -85,B 0,C 180,E1 25971.745,E2 25971.745} C_VEL
LIN {X 0,Y 553.501,Z 619.034,A -85,B 0,C 180,E1 25968.252,E2 25968.252} C_VEL
LIN {X 0,Y 553.493,Z 619.031,A -85,B 0,C 180,E1 25964.914,E2 25964.914} C_VEL
LIN {X 0,Y 553.504,Z 619.038,A -85,B 0,C 180,E1 25961.527,E2 25961.527} C_VEL
LIN {X 0,Y 553.512,Z 619.071,A -85,B 0,C 180,E1 25959.942,E2 25959.942} C_VEL
LIN {X 0,Y 554.565,Z 622.133,A -85,B 0,C 180,E1 25959.493,E2 25959.493} C_VEL
LIN {X 0,Y 555.772,Z 624.767,A -85,B 0,C 180,E1 25959.075,E2 25959.075} C_VEL
LIN {X 0,Y 559.38,Z 632.532,A -85,B 0,C 180,E1 25957.911,E2 25957.911} C_VEL
LIN {X 0,Y 578.265,Z 659.876,A -85,B 0,C 180,E1 25955.809,E2 25955.809} C_VEL
LIN {X 0,Y 585.458,Z 671.186,A -85,B 0,C 180,E1 25955.042,E2 25955.042} C_VEL
LIN {X 0,Y 577.115,Z 912.716,A -85,B 0,C 180,E1 25951.366,E2 25951.366} C_VEL
LIN {X 0,Y 575.601,Z 963.813,A -85,B 0,C 180,E1 25950.571,E2 25950.571} C_VEL
LIN {X 0,Y 574.533,Z 986.671,A -85,B 0,C 180,E1 25950.027,E2 25950.027} C_VEL
LIN {X 0,Y 573.12,Z 1009.771,A -85,B 0,C 180,E1 25949.294,E2 25949.294} C_VEL
LIN {X 0,Y 571.477,Z 1031.606,A -85,B 0,C 180,E1 25948.419,E2 25948.419} C_VEL
LIN {X 0,Y 569.549,Z 1052.433,A -85,B 0,C 180,E1 25947.385,E2 25947.385} C_VEL
LIN {X 0,Y 567.386,Z 1074.003,A -85,B 0,C 180,E1 25946.104,E2 25946.104} C_VEL
LIN {X 0,Y 565.313,Z 1092.847,A -85,B 0,C 180,E1 25944.784,E2 25944.784} C_VEL
LIN {X 0,Y 563.122,Z 1111.232,A -85,B 0,C 180,E1 25943.271,E2 25943.271} C_VEL
LIN {X 0,Y 561.085,Z 1128.323,A -85,B 0,C 180,E1 25941.647,E2 25941.647} C_VEL
LIN {X 0,Y 559.198,Z 1143.523,A -85,B 0,C 180,E1 25939.97,E2 25939.97} C_VEL
LIN {X 0,Y 557.34,Z 1159.193,A -85,B 0,C 180,E1 25937.973,E2 25937.973} C_VEL
LIN {X 0,Y 555.881,Z 1172.005,A -85,B 0,C 180,E1 25936.082,E2 25936.082} C_VEL
LIN {X 0,Y 554.606,Z 1184.149,A -85,B 0,C 180,E1 25933.98,E2 25933.98} C_VEL
LIN {X 0,Y 553.612,Z 1195.043,A -85,B 0,C 180,E1 25931.776,E2 25931.776} C_VEL
LIN {X 0,Y 552.906,Z 1203.984,A -85,B 0,C 180,E1 25929.577,E2 25929.577} C_VEL
LIN {X 0,Y 552.425,Z 1211.993,A -85,B 0,C 180,E1 25927.174,E2 25927.174} C_VEL
LIN {X 0,Y 552.167,Z 1217.691,A -85,B 0,C 180,E1 25924.987,E2 25924.987} C_VEL
LIN {X 0,Y 552.022,Z 1222.461,A -85,B 0,C 180,E1 25922.492,E2 25922.492} C_VEL
LIN {X 0,Y 551.996,Z 1225.32,A -85,B 0,C 180,E1 25920.208,E2 25920.208} C_VEL
LIN {X 0,Y 551.962,Z 1226.663,A -85,B 0,C 180,E1 25917.82,E2 25917.82} C_VEL
LIN {X 0,Y 551.963,Z 1226.581,A -85,B 0,C 180,E1 25915.532,E2 25915.532} C_VEL
LIN {X 0,Y 551.984,Z 1224.909,A -85,B 0,C 180,E1 25913.238,E2 25913.238} C_VEL
LIN {X 0,Y 552.056,Z 1221.878,A -85,B 0,C 180,E1 25910.934,E2 25910.934} C_VEL
LIN {X 0,Y 552.193,Z 1217.407,A -85,B 0,C 180,E1 25908.722,E2 25908.722} C_VEL
LIN {X 0,Y 552.499,Z 1211.148,A -85,B 0,C 180,E1 25906.373,E2 25906.373} C_VEL
LIN {X 0,Y 552.944,Z 1203.968,A -85,B 0,C 180,E1 25904.262,E2 25904.262} C_VEL
LIN {X 0,Y 553.728,Z 1194.153,A -85,B 0,C 180,E1 25901.905,E2 25901.905} C_VEL
LIN {X 0,Y 554.735,Z 1183.396,A -85,B 0,C 180,E1 25899.753,E2 25899.753} C_VEL
LIN {X 0,Y 555.961,Z 1171.094,A -85,B 0,C 180,E1 25897.698,E2 25897.698} C_VEL
LIN {X 0,Y 557.535,Z 1156.657,A -85,B 0,C 180,E1 25895.639,E2 25895.639} C_VEL
LIN {X 0,Y 559.182,Z 1142.052,A -85,B 0,C 180,E1 25893.851,E2 25893.851} C_VEL
LIN {X 0,Y 560.898,Z 1126.395,A -85,B 0,C 180,E1 25892.214,E2 25892.214} C_VEL
LIN {X 0,Y 562.688,Z 1109.586,A -85,B 0,C 180,E1 25890.688,E2 25890.688} C_VEL
LIN {X 0,Y 564.431,Z 1091.873,A -85,B 0,C 180,E1 25889.323,E2 25889.323} C_VEL
LIN {X 0,Y 566.14,Z 1072.672,A -85,B 0,C 180,E1 25888.064,E2 25888.064} C_VEL
LIN {X 0,Y 567.654,Z 1052.963,A -85,B 0,C 180,E1 25886.978,E2 25886.978} C_VEL
LIN {X 0,Y 568.871,Z 1032.747,A -85,B 0,C 180,E1 25886.078,E2 25886.078} C_VEL
LIN {X 0,Y 569.904,Z 1010.752,A -85,B 0,C 180,E1 25885.296,E2 25885.296} C_VEL
LIN {X 0,Y 570.523,Z 990.042,A -85,B 0,C 180,E1 25884.737,E2 25884.737} C_VEL
LIN {X 0,Y 570.789,Z 968.22,A -85,B 0,C 180,E1 25884.333,E2 25884.333} C_VEL
LIN {X 0,Y 572.503,Z 841.331,A -85,B 0,C 180,E1 25882.692,E2 25882.692} C_VEL
LIN {X 0,Y 574.852,Z 746.26,A -85,B 0,C 180,E1 25881.295,E2 25881.295} C_VEL
LIN {X 0,Y 576.308,Z 702.234,A -85,B 0,C 180,E1 25880.584,E2 25880.584} C_VEL
LIN {X 0,Y 572.132,Z 703.449,A -85,B 0,C 180,E1 25880.262,E2 25880.262} C_VEL
LIN {X 0,Y 569.236,Z 703.091,A -85,B 0,C 180,E1 25879.984,E2 25879.984} C_VEL
LIN {X 0,Y 564.761,Z 714.981,A -85,B 0,C 180,E1 25878.573,E2 25878.573} C_VEL
LIN {X 0,Y 561.007,Z 729.991,A -85,B 0,C 180,E1 25877.025,E2 25877.025} C_VEL
LIN {X 0,Y 558.06,Z 748.645,A -85,B 0,C 180,E1 25875.343,E2 25875.343} C_VEL
LIN {X 0,Y 555.843,Z 773.505,A -85,B 0,C 180,E1 25873.344,E2 25873.344} C_VEL
LIN {X 0,Y 555.832,Z 797.22,A -85,B 0,C 180,E1 25871.552,E2 25871.552} C_VEL
LIN {X 0,Y 558.237,Z 818.914,A -85,B 0,C 180,E1 25869.949,E2 25869.949} C_VEL
LIN {X 0,Y 562.458,Z 837.26,A -85,B 0,C 180,E1 25868.608,E2 25868.608} C_VEL
LIN {X 0,Y 568.793,Z 854.863,A -85,B 0,C 180,E1 25867.337,E2 25867.337} C_VEL
LIN {X 0,Y 577.07,Z 871.543,A -85,B 0,C 180,E1 25866.153,E2 25866.153} C_VEL
LIN {X 0,Y 587.103,Z 887.038,A -85,B 0,C 180,E1 25865.081,E2 25865.081} C_VEL
LIN {X 0,Y 596.949,Z 899.419,A -85,B 0,C 180,E1 25864.251,E2 25864.251} C_VEL
LIN {X 0,Y 587.474,Z 912.724,A -85,B 0,C 180,E1 25863.526,E2 25863.526} C_VEL
LIN {X 0,Y 585.204,Z 916.593,A -85,B 0,C 180,E1 25863.33,E2 25863.33} C_VEL
LIN {X 0,Y 578.085,Z 936.679,A -85,B 0,C 180,E1 25863.379,E2 25863.379} C_VEL
LIN {X 0,Y 572.879,Z 956.405,A -85,B 0,C 180,E1 25863.335,E2 25863.335} C_VEL
LIN {X 0,Y 570.522,Z 971.295,A -85,B 0,C 180,E1 25863.168,E2 25863.168} C_VEL
LIN {X 0,Y 568.997,Z 999.726,A -85,B 0,C 180,E1 25862.579,E2 25862.579} C_VEL
LIN {X 0,Y 567.208,Z 1030.442,A -85,B 0,C 180,E1 25861.758,E2 25861.758} C_VEL
LIN {X 0,Y 565.507,Z 1060.222,A -85,B 0,C 180,E1 25860.76,E2 25860.76} C_VEL
LIN {X 0,Y 563.93,Z 1087.501,A -85,B 0,C 180,E1 25859.65,E2 25859.65} C_VEL
LIN {X 0,Y 562.457,Z 1112.3,A -85,B 0,C 180,E1 25858.454,E2 25858.454} C_VEL
LIN {X 0,Y 561.056,Z 1135.488,A -85,B 0,C 180,E1 25857.145,E2 25857.145} C_VEL
LIN {X 0,Y 559.592,Z 1158.713,A -85,B 0,C 180,E1 25855.622,E2 25855.622} C_VEL
LIN {X 0,Y 558.272,Z 1178.578,A -85,B 0,C 180,E1 25854.103,E2 25854.103} C_VEL
LIN {X 0,Y 556.936,Z 1198.046,A -85,B 0,C 180,E1 25852.373,E2 25852.373} C_VEL
LIN {X 0,Y 555.814,Z 1214.731,A -85,B 0,C 180,E1 25850.647,E2 25850.647} C_VEL
LIN {X 0,Y 554.732,Z 1230.678,A -85,B 0,C 180,E1 25848.715,E2 25848.715} C_VEL
LIN {X 0,Y 553.87,Z 1244.198,A -85,B 0,C 180,E1 25846.79,E2 25846.79} C_VEL
LIN {X 0,Y 553.185,Z 1256.178,A -85,B 0,C 180,E1 25844.755,E2 25844.755} C_VEL
LIN {X 0,Y 552.648,Z 1266.561,A -85,B 0,C 180,E1 25842.647,E2 25842.647} C_VEL
LIN {X 0,Y 552.313,Z 1274.968,A -85,B 0,C 180,E1 25840.537,E2 25840.537} C_VEL
LIN {X 0,Y 552.093,Z 1282.203,A -85,B 0,C 180,E1 25838.227,E2 25838.227} C_VEL
LIN {X 0,Y 552.006,Z 1287.059,A -85,B 0,C 180,E1 25836.136,E2 25836.136} C_VEL
LIN {X 0,Y 551.964,Z 1290.494,A -85,B 0,C 180,E1 25834.053,E2 25834.053} C_VEL
LIN {X 0,Y 551.952,Z 1292.631,A -85,B 0,C 180,E1 25831.87,E2 25831.87} C_VEL
LIN {X 0,Y 551.94,Z 1293.169,A -85,B 0,C 180,E1 25829.379,E2 25829.379} C_VEL
LIN {X 0,Y 551.941,Z 1292.073,A -85,B 0,C 180,E1 25827.198,E2 25827.198} C_VEL
LIN {X 0,Y 551.961,Z 1289.404,A -85,B 0,C 180,E1 25824.909,E2 25824.909} C_VEL
LIN {X 0,Y 552.025,Z 1284.573,A -85,B 0,C 180,E1 25822.403,E2 25822.403} C_VEL
LIN {X 0,Y 552.194,Z 1278.64,A -85,B 0,C 180,E1 25820.201,E2 25820.201} C_VEL
LIN {X 0,Y 552.511,Z 1271.109,A -85,B 0,C 180,E1 25817.99,E2 25817.99} C_VEL
LIN {X 0,Y 553.035,Z 1261.291,A -85,B 0,C 180,E1 25815.66,E2 25815.66} C_VEL
LIN {X 0,Y 553.805,Z 1249.893,A -85,B 0,C 180,E1 25813.427,E2 25813.427} C_VEL
LIN {X 0,Y 554.908,Z 1236.358,A -85,B 0,C 180,E1 25811.185,E2 25811.185} C_VEL
LIN {X 0,Y 556.38,Z 1220.333,A -85,B 0,C 180,E1 25808.937,E2 25808.937} C_VEL
LIN {X 0,Y 558.072,Z 1203.343,A -85,B 0,C 180,E1 25806.899,E2 25806.899} C_VEL
LIN {X 0,Y 559.926,Z 1185.806,A -85,B 0,C 180,E1 25805.077,E2 25805.077} C_VEL
LIN {X 0,Y 562.196,Z 1165.247,A -85,B 0,C 180,E1 25803.231,E2 25803.231} C_VEL
LIN {X 0,Y 564.409,Z 1145.329,A -85,B 0,C 180,E1 25801.7,E2 25801.7} C_VEL
LIN {X 0,Y 566.796,Z 1124.308,A -85,B 0,C 180,E1 25800.285,E2 25800.285} C_VEL
LIN {X 0,Y 569.11,Z 1103.081,A -85,B 0,C 180,E1 25799.078,E2 25799.078} C_VEL
LIN {X 0,Y 571.532,Z 1080.771,A -85,B 0,C 180,E1 25797.99,E2 25797.99} C_VEL
LIN {X 0,Y 573.848,Z 1057.643,A -85,B 0,C 180,E1 25797.071,E2 25797.071} C_VEL
LIN {X 0,Y 576.1,Z 1033.992,A -85,B 0,C 180,E1 25796.302,E2 25796.302} C_VEL
LIN {X 0,Y 578.059,Z 1009.928,A -85,B 0,C 180,E1 25795.718,E2 25795.718} C_VEL
LIN {X 0,Y 579.466,Z 984.915,A -85,B 0,C 180,E1 25795.254,E2 25795.254} C_VEL
LIN {X 0,Y 580.677,Z 967.598,A -85,B 0,C 180,E1 25795.02,E2 25795.02} C_VEL
LIN {X 0,Y 582.578,Z 954.556,A -85,B 0,C 180,E1 25794.905,E2 25794.905} C_VEL
LIN {X 0,Y 590.395,Z 940.948,A -85,B 0,C 180,E1 25794.19,E2 25794.19} C_VEL
LIN {X 0,Y 601.586,Z 923.668,A -85,B 0,C 180,E1 25793.369,E2 25793.369} C_VEL
LIN {X 0,Y 604.628,Z 919.203,A -85,B 0,C 180,E1 25793.169,E2 25793.169} C_VEL
LIN {X 0,Y 595.051,Z 908.005,A -85,B 0,C 180,E1 25791.695,E2 25791.695} C_VEL
LIN {X 0,Y 587.325,Z 895.323,A -85,B 0,C 180,E1 25790.157,E2 25790.157} C_VEL
LIN {X 0,Y 581.432,Z 881.023,A -85,B 0,C 180,E1 25788.543,E2 25788.543} C_VEL
LIN {X 0,Y 577.659,Z 865.63,A -85,B 0,C 180,E1 25786.925,E2 25786.925} C_VEL
LIN {X 0,Y 575.933,Z 848.35,A -85,B 0,C 180,E1 25785.241,E2 25785.241} C_VEL
LIN {X 0,Y 576.33,Z 828.464,A -85,B 0,C 180,E1 25783.438,E2 25783.438} C_VEL
LIN {X 0,Y 579.927,Z 789.285,A -85,B 0,C 180,E1 25780.025,E2 25780.025} C_VEL
LIN {X 0,Y 583.33,Z 753.844,A -85,B 0,C 180,E1 25776.866,E2 25776.866} C_VEL
LIN {X 0,Y 586.649,Z 719.861,A -85,B 0,C 180,E1 25773.755,E2 25773.755} C_VEL
LIN {X 0,Y 588.57,Z 698.862,A -85,B 0,C 180,E1 25771.779,E2 25771.779} C_VEL
LIN {X 0,Y 580.502,Z 679.269,A -85,B 0,C 180,E1 25768.835,E2 25768.835} C_VEL
LIN {X 0,Y 573.101,Z 662.221,A -85,B 0,C 180,E1 25766.083,E2 25766.083} C_VEL
LIN {X 0,Y 566.414,Z 647.261,A -85,B 0,C 180,E1 25763.513,E2 25763.513} C_VEL
LIN {X 0,Y 560.581,Z 634.768,A -85,B 0,C 180,E1 25761.228,E2 25761.228} C_VEL
LIN {X 0,Y 556.908,Z 626.89,A -85,B 0,C 180,E1 25759.727,E2 25759.727} C_VEL
LIN {X 0,Y 554.966,Z 622.756,A -85,B 0,C 180,E1 25758.924,E2 25758.924} C_VEL
LIN {X 0,Y 553.541,Z 619.316,A -85,B 0,C 180,E1 25758.264,E2 25758.264} C_VEL
LIN {X 0,Y 553.501,Z 619.038,A -85,B 0,C 180,E1 25757.994,E2 25757.994} C_VEL
LIN {X 0,Y 553.505,Z 619.03,A -85,B 0,C 180,E1 25754.65,E2 25754.65} C_VEL
LIN {X 0,Y 553.493,Z 619.03,A -85,B 0,C 180,E1 25751.251,E2 25751.251} C_VEL
LIN {X 0,Y 553.507,Z 619.032,A -85,B 0,C 180,E1 25747.787,E2 25747.787} C_VEL
LIN {X 0,Y 553.489,Z 619.035,A -85,B 0,C 180,E1 25744.351,E2 25744.351} C_VEL
LIN {X 0,Y 553.486,Z 619.029,A -85,B 0,C 180,E1 25741.035,E2 25741.035} C_VEL
LIN {X 0,Y 553.486,Z 619.031,A -85,B 0,C 180,E1 25737.826,E2 25737.826} C_VEL
LIN {X 0,Y 553.496,Z 619.035,A -85,B 0,C 180,E1 25734.467,E2 25734.467} C_VEL
LIN {X 0,Y 553.504,Z 619.036,A -85,B 0,C 180,E1 25731.153,E2 25731.153} C_VEL
LIN {X 0,Y 553.504,Z 619.035,A -85,B 0,C 180,E1 25727.758,E2 25727.758} C_VEL
LIN {X 0,Y 553.492,Z 619.034,A -85,B 0,C 180,E1 25724.385,E2 25724.385} C_VEL
LIN {X 0,Y 553.506,Z 619.032,A -85,B 0,C 180,E1 25721.024,E2 25721.024} C_VEL
LIN {X 0,Y 553.507,Z 619.032,A -85,B 0,C 180,E1 25717.594,E2 25717.594} C_VEL
LIN {X 0,Y 553.494,Z 619.035,A -85,B 0,C 180,E1 25714.191,E2 25714.191} C_VEL
LIN {X 0,Y 553.488,Z 619.035,A -85,B 0,C 180,E1 25710.925,E2 25710.925} C_VEL
LIN {X 0,Y 553.489,Z 619.033,A -85,B 0,C 180,E1 25707.674,E2 25707.674} C_VEL
LIN {X 0,Y 553.492,Z 619.028,A -85,B 0,C 180,E1 25704.38,E2 25704.38} C_VEL
LIN {X 0,Y 553.511,Z 619.026,A -85,B 0,C 180,E1 25700.916,E2 25700.916} C_VEL
LIN {X 0,Y 553.499,Z 619.012,A -85,B 0,C 180,E1 25697.631,E2 25697.631} C_VEL
LIN {X 0,Y 553.504,Z 619.036,A -85,B 0,C 180,E1 25694.208,E2 25694.208} C_VEL
LIN {X 0,Y 553.495,Z 619.019,A -85,B 0,C 180,E1 25690.806,E2 25690.806} C_VEL
LIN {X 0,Y 553.501,Z 619.019,A -85,B 0,C 180,E1 25687.358,E2 25687.358} C_VEL
LIN {X 0,Y 553.499,Z 619.117,A -85,B 0,C 180,E1 25685.926,E2 25685.926} C_VEL
LIN {X 0,Y 562.267,Z 644.489,A -85,B 0,C 180,E1 25683.575,E2 25683.575} C_VEL
LIN {X 0,Y 566.849,Z 660.036,A -85,B 0,C 180,E1 25682.187,E2 25682.187} C_VEL
LIN {X 0,Y 565.367,Z 702.845,A -85,B 0,C 180,E1 25679.099,E2 25679.099} C_VEL
LIN {X 0,Y 563.491,Z 749.321,A -85,B 0,C 180,E1 25675.712,E2 25675.712} C_VEL
LIN {X 0,Y 561.715,Z 797.205,A -85,B 0,C 180,E1 25672.279,E2 25672.279} C_VEL
LIN {X 0,Y 560.915,Z 824.096,A -85,B 0,C 180,E1 25670.417,E2 25670.417} C_VEL
LIN {X 0,Y 559.934,Z 830.64,A -85,B 0,C 180,E1 25670.01,E2 25670.01} C_VEL
LIN {X 0,Y 556.955,Z 840.341,A -85,B 0,C 180,E1 25669.552,E2 25669.552} C_VEL
LIN {X 0,Y 554.439,Z 849.569,A -85,B 0,C 180,E1 25669.267,E2 25669.267} C_VEL
LIN {X 0,Y 553.745,Z 856.037,A -85,B 0,C 180,E1 25669.148,E2 25669.148} C_VEL
LIN {X 0,Y 551.919,Z 1015.476,A -85,B 0,C 180,E1 25667.031,E2 25667.031} C_VEL
LIN {X 0,Y 551.666,Z 1033.048,A -85,B 0,C 180,E1 25666.609,E2 25666.609} C_VEL
LIN {X 0,Y 551.171,Z 1049.749,A -85,B 0,C 180,E1 25666.005,E2 25666.005} C_VEL
LIN {X 0,Y 550.496,Z 1065.976,A -85,B 0,C 180,E1 25665.214,E2 25665.214} C_VEL
LIN {X 0,Y 549.701,Z 1081.148,A -85,B 0,C 180,E1 25664.267,E2 25664.267} C_VEL
LIN {X 0,Y 548.834,Z 1095.228,A -85,B 0,C 180,E1 25663.162,E2 25663.162} C_VEL
LIN {X 0,Y 547.943,Z 1108.236,A -85,B 0,C 180,E1 25661.898,E2 25661.898} C_VEL
LIN {X 0,Y 547.1,Z 1119.994,A -85,B 0,C 180,E1 25660.497,E2 25660.497} C_VEL
LIN {X 0,Y 546.39,Z 1129.845,A -85,B 0,C 180,E1 25659.053,E2 25659.053} C_VEL
LIN {X 0,Y 545.784,Z 1138.493,A -85,B 0,C 180,E1 25657.472,E2 25657.472} C_VEL
LIN {X 0,Y 545.318,Z 1145.696,A -85,B 0,C 180,E1 25655.786,E2 25655.786} C_VEL
LIN {X 0,Y 544.992,Z 1151.397,A -85,B 0,C 180,E1 25653.996,E2 25653.996} C_VEL
LIN {X 0,Y 544.799,Z 1155.288,A -85,B 0,C 180,E1 25652.207,E2 25652.207} C_VEL
LIN {X 0,Y 544.704,Z 1157.509,A -85,B 0,C 180,E1 25650.314,E2 25650.314} C_VEL
LIN {X 0,Y 544.684,Z 1157.936,A -85,B 0,C 180,E1 25648.421,E2 25648.421} C_VEL
LIN {X 0,Y 544.756,Z 1156.586,A -85,B 0,C 180,E1 25646.526,E2 25646.526} C_VEL
LIN {X 0,Y 544.909,Z 1153.562,A -85,B 0,C 180,E1 25644.734,E2 25644.734} C_VEL
LIN {X 0,Y 545.186,Z 1148.767,A -85,B 0,C 180,E1 25642.94,E2 25642.94} C_VEL
LIN {X 0,Y 545.613,Z 1142.078,A -85,B 0,C 180,E1 25641.143,E2 25641.143} C_VEL
LIN {X 0,Y 546.161,Z 1134.358,A -85,B 0,C 180,E1 25639.556,E2 25639.556} C_VEL
LIN {X 0,Y 546.883,Z 1124.549,A -85,B 0,C 180,E1 25637.968,E2 25637.968} C_VEL
LIN {X 0,Y 547.739,Z 1113.168,A -85,B 0,C 180,E1 25636.486,E2 25636.486} C_VEL
LIN {X 0,Y 548.639,Z 1100.781,A -85,B 0,C 180,E1 25635.175,E2 25635.175} C_VEL
LIN {X 0,Y 549.55,Z 1087.03,A -85,B 0,C 180,E1 25633.998,E2 25633.998} C_VEL
LIN {X 0,Y 550.388,Z 1072.418,A -85,B 0,C 180,E1 25632.992,E2 25632.992} C_VEL
LIN {X 0,Y 551.131,Z 1056.85,A -85,B 0,C 180,E1 25632.144,E2 25632.144} C_VEL
LIN {X 0,Y 551.733,Z 1040.167,A -85,B 0,C 180,E1 25631.454,E2 25631.454} C_VEL
LIN {X 0,Y 552.101,Z 1022.796,A -85,B 0,C 180,E1 25630.953,E2 25630.953} C_VEL
LIN {X 0,Y 552.245,Z 1003.32,A -85,B 0,C 180,E1 25630.612,E2 25630.612} C_VEL
LIN {X 0,Y 553.908,Z 850.241,A -85,B 0,C 180,E1 25628.594,E2 25628.594} C_VEL
LIN {X 0,Y 553.254,Z 845.093,A -85,B 0,C 180,E1 25628.476,E2 25628.476} C_VEL
LIN {X 0,Y 554.573,Z 799.516,A -85,B 0,C 180,E1 25625.328,E2 25625.328} C_VEL
LIN {X 0,Y 556.384,Z 753.915,A -85,B 0,C 180,E1 25622.026,E2 25622.026} C_VEL
LIN {X 0,Y 558.394,Z 707.151,A -85,B 0,C 180,E1 25618.594,E2 25618.594} C_VEL
LIN {X 0,Y 559.944,Z 667.62,A -85,B 0,C 180,E1 25615.709,E2 25615.709} C_VEL
LIN {X 0,Y 559.932,Z 662.381,A -85,B 0,C 180,E1 25615.319,E2 25615.319} C_VEL
LIN {X 0,Y 552.774,Z 639.934,A -85,B 0,C 180,E1 25613.22,E2 25613.22} C_VEL
LIN {X 0,Y 545.566,Z 620.012,A -85,B 0,C 180,E1 25611.285,E2 25611.285} C_VEL
LIN {X 0,Y 545.551,Z 620.025,A -85,B 0,C 180,E1 25607.927,E2 25607.927} C_VEL
LIN {X 0,Y 545.554,Z 620.019,A -85,B 0,C 180,E1 25604.585,E2 25604.585} C_VEL
LIN {X 0,Y 545.575,Z 620.021,A -85,B 0,C 180,E1 25601.126,E2 25601.126} C_VEL
LIN {X 0,Y 545.59,Z 620.29,A -85,B 0,C 180,E1 25600.726,E2 25600.726} C_VEL
LIN {X 0,Y 547.045,Z 623.759,A -85,B 0,C 180,E1 25600.179,E2 25600.179} C_VEL
LIN {X 0,Y 551.931,Z 634.503,A -85,B 0,C 180,E1 25598.528,E2 25598.528} C_VEL
LIN {X 0,Y 569.936,Z 660.456,A -85,B 0,C 180,E1 25596.469,E2 25596.469} C_VEL
LIN {X 0,Y 579.011,Z 674.465,A -85,B 0,C 180,E1 25595.478,E2 25595.478} C_VEL
LIN {X 0,Y 570.223,Z 914.354,A -85,B 0,C 180,E1 25591.758,E2 25591.758} C_VEL
LIN {X 0,Y 568.617,Z 965.062,A -85,B 0,C 180,E1 25590.949,E2 25590.949} C_VEL
LIN {X 0,Y 567.503,Z 988.062,A -85,B 0,C 180,E1 25590.391,E2 25590.391} C_VEL
LIN {X 0,Y 566.017,Z 1011.218,A -85,B 0,C 180,E1 25589.64,E2 25589.64} C_VEL
LIN {X 0,Y 564.311,Z 1032.918,A -85,B 0,C 180,E1 25588.755,E2 25588.755} C_VEL
LIN {X 0,Y 562.321,Z 1053.662,A -85,B 0,C 180,E1 25587.709,E2 25587.709} C_VEL
LIN {X 0,Y 560.047,Z 1075.416,A -85,B 0,C 180,E1 25586.395,E2 25586.395} C_VEL
LIN {X 0,Y 557.928,Z 1093.933,A -85,B 0,C 180,E1 25585.078,E2 25585.078} C_VEL
LIN {X 0,Y 555.648,Z 1112.237,A -85,B 0,C 180,E1 25583.546,E2 25583.546} C_VEL
LIN {X 0,Y 553.461,Z 1129.77,A -85,B 0,C 180,E1 25581.849,E2 25581.849} C_VEL
LIN {X 0,Y 551.428,Z 1145.606,A -85,B 0,C 180,E1 25580.068,E2 25580.068} C_VEL
LIN {X 0,Y 549.579,Z 1160.458,A -85,B 0,C 180,E1 25578.126,E2 25578.126} C_VEL
LIN {X 0,Y 547.998,Z 1173.879,A -85,B 0,C 180,E1 25576.102,E2 25576.102} C_VEL
LIN {X 0,Y 546.678,Z 1185.795,A -85,B 0,C 180,E1 25573.971,E2 25573.971} C_VEL
LIN {X 0,Y 545.651,Z 1196.473,A -85,B 0,C 180,E1 25571.736,E2 25571.736} C_VEL
LIN {X 0,Y 544.963,Z 1204.913,A -85,B 0,C 180,E1 25569.611,E2 25569.611} C_VEL
LIN {X 0,Y 544.459,Z 1212.816,A -85,B 0,C 180,E1 25567.174,E2 25567.174} C_VEL
LIN {X 0,Y 544.192,Z 1218.465,A -85,B 0,C 180,E1 25564.954,E2 25564.954} C_VEL
LIN {X 0,Y 544.043,Z 1222.974,A -85,B 0,C 180,E1 25562.528,E2 25562.528} C_VEL
LIN {X 0,Y 544.012,Z 1225.825,A -85,B 0,C 180,E1 25560.211,E2 25560.211} C_VEL
LIN {X 0,Y 543.978,Z 1227.124,A -85,B 0,C 180,E1 25557.893,E2 25557.893} C_VEL
LIN {X 0,Y 543.978,Z 1227.097,A -85,B 0,C 180,E1 25555.678,E2 25555.678} C_VEL
LIN {X 0,Y 543.995,Z 1225.559,A -85,B 0,C 180,E1 25553.35,E2 25553.35} C_VEL
LIN {X 0,Y 544.073,Z 1222.635,A -85,B 0,C 180,E1 25551.013,E2 25551.013} C_VEL
LIN {X 0,Y 544.229,Z 1218.012,A -85,B 0,C 180,E1 25548.663,E2 25548.663} C_VEL
